LIN {X 0,Y 525.118,Z 322.281,A -85,B 0,C 180,E1 -4783.004,E2 -4783.004} C_VEL
LIN {X 0,Y 525.376,Z 308.759,A -85,B 0,C 180,E1 -4783.44,E2 -4783.44} C_VEL
LIN {X 0,Y 525.556,Z 295.266,A -85,B 0,C 180,E1 -4783.706,E2 -4783.706} C_VEL
LIN {X 0,Y 525.721,Z 203.156,A -85,B 0,C 180,E1 -4784.977,E2 -4784.977} C_VEL
LIN {X 0,Y 524.2,Z 193.139,A -85,B 0,C 180,E1 -4785.174,E2 -4785.174} C_VEL
LIN {X 0,Y 524.565,Z 174.875,A -85,B 0,C 180,E1 -4787.948,E2 -4787.948} C_VEL
LIN {X 0,Y 524.995,Z 155.161,A -85,B 0,C 180,E1 -4790.983,E2 -4790.983} C_VEL
LIN {X 0,Y 525.282,Z 140.673,A -85,B 0,C 180,E1 -4793.247,E2 -4793.247} C_VEL
LIN {X 0,Y 523.943,Z 133.222,A -85,B 0,C 180,E1 -4794.518,E2 -4794.518} C_VEL
LIN {X 0,Y 523.92,Z 133.229,A -85,B 0,C 180,E1 -4797.706,E2 -4797.706} C_VEL
LIN {X 0,Y 523.946,Z 133.218,A -85,B 0,C 180,E1 -4800.645,E2 -4800.645} C_VEL
LIN {X 0,Y 523.928,Z 133.222,A -85,B 0,C 180,E1 -4803.729,E2 -4803.729} C_VEL
LIN {X 0,Y 523.889,Z 133.223,A -85,B 0,C 180,E1 -4806.399,E2 -4806.399} C_VEL
LIN {X 0,Y 523.911,Z 133.226,A -85,B 0,C 180,E1 -4809.086,E2 -4809.086} C_VEL
LIN {X 0,Y 523.893,Z 133.223,A -85,B 0,C 180,E1 -4812.125,E2 -4812.125} C_VEL
LIN {X 0,Y 523.936,Z 133.223,A -85,B 0,C 180,E1 -4815.311,E2 -4815.311} C_VEL
LIN {X 0,Y 523.911,Z 133.225,A -85,B 0,C 180,E1 -4818.696,E2 -4818.696} C_VEL
LIN {X 0,Y 523.88,Z 133.223,A -85,B 0,C 180,E1 -4821.895,E2 -4821.895} C_VEL
LIN {X 0,Y 523.887,Z 133.228,A -85,B 0,C 180,E1 -4824.917,E2 -4824.917} C_VEL
LIN {X 0,Y 523.9,Z 133.221,A -85,B 0,C 180,E1 -4827.686,E2 -4827.686} C_VEL
LIN {X 0,Y 523.868,Z 133.227,A -85,B 0,C 180,E1 -4830.239,E2 -4830.239} C_VEL
LIN {X 0,Y 523.894,Z 133.223,A -85,B 0,C 180,E1 -4832.863,E2 -4832.863} C_VEL
LIN {X 0,Y 523.913,Z 133.221,A -85,B 0,C 180,E1 -4835.809,E2 -4835.809} C_VEL
LIN {X 0,Y 523.901,Z 133.224,A -85,B 0,C 180,E1 -4838.764,E2 -4838.764} C_VEL
LIN {X 0,Y 523.899,Z 133.22,A -85,B 0,C 180,E1 -4841.218,E2 -4841.218} C_VEL
LIN {X 0,Y 523.881,Z 133.224,A -85,B 0,C 180,E1 -4843.637,E2 -4843.637} C_VEL
LIN {X 0,Y 523.916,Z 133.226,A -85,B 0,C 180,E1 -4846.027,E2 -4846.027} C_VEL
LIN {X 0,Y 523.964,Z 133.217,A -85,B 0,C 180,E1 -4848.393,E2 -4848.393} C_VEL
LIN {X 0,Y 523.957,Z 133.216,A -85,B 0,C 180,E1 -4851.515,E2 -4851.515} C_VEL
LIN {X 0,Y 524.037,Z 133.204,A -85,B 0,C 180,E1 -4854.613,E2 -4854.613} C_VEL
LIN {X 0,Y 524.108,Z 133.2,A -85,B 0,C 180,E1 -4857.694,E2 -4857.694} C_VEL
LIN {X 0,Y 524.103,Z 133.198,A -85,B 0,C 180,E1 -4860,E2 -4860} C_VEL
LIN {X 0,Y 524.038,Z 133.205,A -85,B 0,C 180,E1 -4863.075,E2 -4863.075} C_VEL
LIN {X 0,Y 524.014,Z 133.205,A -85,B 0,C 180,E1 -4866.159,E2 -4866.159} C_VEL
LIN {X 0,Y 523.985,Z 133.218,A -85,B 0,C 180,E1 -4869.262,E2 -4869.262} C_VEL
LIN {X 0,Y 524.002,Z 133.211,A -85,B 0,C 180,E1 -4871.737,E2 -4871.737} C_VEL
LIN {X 0,Y 523.993,Z 133.214,A -85,B 0,C 180,E1 -4875.051,E2 -4875.051} C_VEL
LIN {X 0,Y 523.946,Z 133.214,A -85,B 0,C 180,E1 -4877.969,E2 -4877.969} C_VEL
LIN {X 0,Y 523.973,Z 133.214,A -85,B 0,C 180,E1 -4880.409,E2 -4880.409} C_VEL
LIN {X 0,Y 523.909,Z 133.227,A -85,B 0,C 180,E1 -4882.893,E2 -4882.893} C_VEL
LIN {X 0,Y 523.916,Z 133.221,A -85,B 0,C 180,E1 -4885.42,E2 -4885.42} C_VEL
LIN {X 0,Y 523.965,Z 133.214,A -85,B 0,C 180,E1 -4887.999,E2 -4887.999} C_VEL
LIN {X 0,Y 523.939,Z 133.223,A -85,B 0,C 180,E1 -4890.853,E2 -4890.853} C_VEL
LIN {X 0,Y 523.93,Z 133.218,A -85,B 0,C 180,E1 -4893.729,E2 -4893.729} C_VEL
LIN {X 0,Y 523.903,Z 133.23,A -85,B 0,C 180,E1 -4896.401,E2 -4896.401} C_VEL
LIN {X 0,Y 523.919,Z 133.221,A -85,B 0,C 180,E1 -4899.084,E2 -4899.084} C_VEL
LIN {X 0,Y 523.953,Z 133.222,A -85,B 0,C 180,E1 -4902.118,E2 -4902.118} C_VEL
LIN {X 0,Y 523.954,Z 133.217,A -85,B 0,C 180,E1 -4905.308,E2 -4905.308} C_VEL
LIN {X 0,Y 523.917,Z 133.222,A -85,B 0,C 180,E1 -4906.875,E2 -4906.875} C_VEL
LIN {X 0,Y 523.237,Z 133.308,A -85,B 0,C 180,E1 -4907.303,E2 -4907.303} C_VEL
LIN {X 0,Y 520.4,Z 133.666,A -85,B 0,C 180,E1 -4907.972,E2 -4907.972} C_VEL
LIN {X 0,Y 517.561,Z 134.017,A -85,B 0,C 180,E1 -4908.648,E2 -4908.648} C_VEL
LIN {X 0,Y 516.896,Z 134.098,A -85,B 0,C 180,E1 -4909.083,E2 -4909.083} C_VEL
LIN {X 0,Y 516.919,Z 134.178,A -85,B 0,C 180,E1 -4910.156,E2 -4910.156} C_VEL
LIN {X 0,Y 517.564,Z 138.657,A -85,B 0,C 180,E1 -4911.044,E2 -4911.044} C_VEL
LIN {X 0,Y 517.333,Z 154.345,A -85,B 0,C 180,E1 -4914.016,E2 -4914.016} C_VEL
LIN {X 0,Y 517.252,Z 157.921,A -85,B 0,C 180,E1 -4914.692,E2 -4914.692} C_VEL
LIN {X 0,Y 519.187,Z 168.539,A -85,B 0,C 180,E1 -4914.905,E2 -4914.905} C_VEL
LIN {X 0,Y 518.635,Z 265.409,A -85,B 0,C 180,E1 -4916.278,E2 -4916.278} C_VEL
LIN {X 0,Y 518.463,Z 278.587,A -85,B 0,C 180,E1 -4916.629,E2 -4916.629} C_VEL
LIN {X 0,Y 518.178,Z 291.605,A -85,B 0,C 180,E1 -4917.145,E2 -4917.145} C_VEL
LIN {X 0,Y 517.868,Z 303.866,A -85,B 0,C 180,E1 -4917.814,E2 -4917.814} C_VEL
LIN {X 0,Y 517.604,Z 314.805,A -85,B 0,C 180,E1 -4918.58,E2 -4918.58} C_VEL
LIN {X 0,Y 517.326,Z 325.178,A -85,B 0,C 180,E1 -4919.486,E2 -4919.486} C_VEL
LIN {X 0,Y 517.019,Z 334.784,A -85,B 0,C 180,E1 -4920.531,E2 -4920.531} C_VEL
LIN {X 0,Y 516.781,Z 343.741,A -85,B 0,C 180,E1 -4921.738,E2 -4921.738} C_VEL
LIN {X 0,Y 516.573,Z 350.564,A -85,B 0,C 180,E1 -4922.886,E2 -4922.886} C_VEL
LIN {X 0,Y 516.437,Z 356.66,A -85,B 0,C 180,E1 -4924.184,E2 -4924.184} C_VEL
LIN {X 0,Y 516.345,Z 361.243,A -85,B 0,C 180,E1 -4925.452,E2 -4925.452} C_VEL
LIN {X 0,Y 516.233,Z 364.666,A -85,B 0,C 180,E1 -4926.746,E2 -4926.746} C_VEL
LIN {X 0,Y 516.2,Z 366.557,A -85,B 0,C 180,E1 -4927.789,E2 -4927.789} C_VEL
LIN {X 0,Y 516.187,Z 368.012,A -85,B 0,C 180,E1 -4929.268,E2 -4929.268} C_VEL
LIN {X 0,Y 516.215,Z 368.215,A -85,B 0,C 180,E1 -4930.101,E2 -4930.101} C_VEL
LIN {X 0,Y 516.174,Z 367.944,A -85,B 0,C 180,E1 -4930.927,E2 -4930.927} C_VEL
LIN {X 0,Y 516.231,Z 366.456,A -85,B 0,C 180,E1 -4932.359,E2 -4932.359} C_VEL
LIN {X 0,Y 516.28,Z 363.606,A -85,B 0,C 180,E1 -4933.796,E2 -4933.796} C_VEL
LIN {X 0,Y 516.419,Z 359.814,A -85,B 0,C 180,E1 -4935.069,E2 -4935.069} C_VEL
LIN {X 0,Y 516.474,Z 355.286,A -85,B 0,C 180,E1 -4936.224,E2 -4936.224} C_VEL
LIN {X 0,Y 516.639,Z 349.277,A -85,B 0,C 180,E1 -4937.429,E2 -4937.429} C_VEL
LIN {X 0,Y 516.828,Z 341.473,A -85,B 0,C 180,E1 -4938.677,E2 -4938.677} C_VEL
LIN {X 0,Y 517.054,Z 332.52,A -85,B 0,C 180,E1 -4939.822,E2 -4939.822} C_VEL
LIN {X 0,Y 517.364,Z 322.862,A -85,B 0,C 180,E1 -4940.816,E2 -4940.816} C_VEL
LIN {X 0,Y 517.716,Z 311.758,A -85,B 0,C 180,E1 -4941.737,E2 -4941.737} C_VEL
LIN {X 0,Y 518.039,Z 300.296,A -85,B 0,C 180,E1 -4942.484,E2 -4942.484} C_VEL
LIN {X 0,Y 518.266,Z 287.201,A -85,B 0,C 180,E1 -4943.137,E2 -4943.137} C_VEL
LIN {X 0,Y 518.467,Z 274.863,A -85,B 0,C 180,E1 -4943.579,E2 -4943.579} C_VEL
LIN {X 0,Y 518.668,Z 261.95,A -85,B 0,C 180,E1 -4943.875,E2 -4943.875} C_VEL
LIN {X 0,Y 518.988,Z 167.401,A -85,B 0,C 180,E1 -4945.206,E2 -4945.206} C_VEL
LIN {X 0,Y 517.232,Z 157.733,A -85,B 0,C 180,E1 -4945.421,E2 -4945.421} C_VEL
LIN {X 0,Y 517.496,Z 141.997,A -85,B 0,C 180,E1 -4948.444,E2 -4948.444} C_VEL
LIN {X 0,Y 517.288,Z 135.99,A -85,B 0,C 180,E1 -4949.611,E2 -4949.611} C_VEL
LIN {X 0,Y 517.061,Z 134.082,A -85,B 0,C 180,E1 -4950,E2 -4950} C_VEL
LIN {X 0,Y 517.068,Z 134.08,A -85,B 0,C 180,E1 -4952.337,E2 -4952.337} C_VEL
LIN {X 0,Y 516.963,Z 134.089,A -85,B 0,C 180,E1 -4956.244,E2 -4956.244} C_VEL
LIN {X 0,Y 516.901,Z 134.095,A -85,B 0,C 180,E1 -4959.39,E2 -4959.39} C_VEL
LIN {X 0,Y 516.881,Z 134.095,A -85,B 0,C 180,E1 -4962.565,E2 -4962.565} C_VEL
LIN {X 0,Y 516.887,Z 134.096,A -85,B 0,C 180,E1 -4965.124,E2 -4965.124} C_VEL
LIN {X 0,Y 516.841,Z 134.101,A -85,B 0,C 180,E1 -4968.226,E2 -4968.226} C_VEL
LIN {X 0,Y 516.858,Z 134.098,A -85,B 0,C 180,E1 -4970.704,E2 -4970.704} C_VEL
LIN {X 0,Y 516.833,Z 134.106,A -85,B 0,C 180,E1 -4973.226,E2 -4973.226} C_VEL
LIN {X 0,Y 516.854,Z 134.099,A -85,B 0,C 180,E1 -4976.177,E2 -4976.177} C_VEL
LIN {X 0,Y 516.825,Z 134.102,A -85,B 0,C 180,E1 -4978.421,E2 -4978.421} C_VEL
LIN {X 0,Y 516.844,Z 134.106,A -85,B 0,C 180,E1 -4981.113,E2 -4981.113} C_VEL
LIN {X 0,Y 516.865,Z 134.098,A -85,B 0,C 180,E1 -4983.96,E2 -4983.96} C_VEL
LIN {X 0,Y 516.803,Z 134.108,A -85,B 0,C 180,E1 -4986.753,E2 -4986.753} C_VEL
LIN {X 0,Y 516.851,Z 134.1,A -85,B 0,C 180,E1 -4989.725,E2 -4989.725} C_VEL
LIN {X 0,Y 516.839,Z 134.107,A -85,B 0,C 180,E1 -4992.837,E2 -4992.837} C_VEL
LIN {X 0,Y 516.895,Z 134.102,A -85,B 0,C 180,E1 -4995.008,E2 -4995.008} C_VEL
LIN {X 0,Y 516.846,Z 134.102,A -85,B 0,C 180,E1 -4998.408,E2 -4998.408} C_VEL
LIN {X 0,Y 516.868,Z 134.099,A -85,B 0,C 180,E1 -5001.284,E2 -5001.284} C_VEL
LIN {X 0,Y 516.849,Z 134.108,A -85,B 0,C 180,E1 -5004.674,E2 -5004.674} C_VEL
LIN {X 0,Y 516.864,Z 134.097,A -85,B 0,C 180,E1 -5007.463,E2 -5007.463} C_VEL
LIN {X 0,Y 516.839,Z 134.108,A -85,B 0,C 180,E1 -5010.492,E2 -5010.492} C_VEL
LIN {X 0,Y 516.831,Z 134.101,A -85,B 0,C 180,E1 -5013.338,E2 -5013.338} C_VEL
LIN {X 0,Y 516.867,Z 134.099,A -85,B 0,C 180,E1 -5015.926,E2 -5015.926} C_VEL
LIN {X 0,Y 516.852,Z 134.106,A -85,B 0,C 180,E1 -5018.461,E2 -5018.461} C_VEL
LIN {X 0,Y 516.848,Z 134.1,A -85,B 0,C 180,E1 -5020.953,E2 -5020.953} C_VEL
LIN {X 0,Y 516.834,Z 134.101,A -85,B 0,C 180,E1 -5023.408,E2 -5023.408} C_VEL
LIN {X 0,Y 516.857,Z 134.102,A -85,B 0,C 180,E1 -5025.833,E2 -5025.833} C_VEL
LIN {X 0,Y 516.928,Z 134.097,A -85,B 0,C 180,E1 -5028.233,E2 -5028.233} C_VEL
LIN {X 0,Y 516.923,Z 134.091,A -85,B 0,C 180,E1 -5031.399,E2 -5031.399} C_VEL
LIN {X 0,Y 516.982,Z 134.084,A -85,B 0,C 180,E1 -5034.54,E2 -5034.54} C_VEL
LIN {X 0,Y 517.076,Z 134.076,A -85,B 0,C 180,E1 -5037.664,E2 -5037.664} C_VEL
LIN {X 0,Y 517.069,Z 134.078,A -85,B 0,C 180,E1 -5040,E2 -5040} C_VEL
LIN {X 0,Y 517.076,Z 134.073,A -85,B 0,C 180,E1 -5042.337,E2 -5042.337} C_VEL
LIN {X 0,Y 516.983,Z 134.088,A -85,B 0,C 180,E1 -5045.461,E2 -5045.461} C_VEL
LIN {X 0,Y 516.925,Z 134.09,A -85,B 0,C 180,E1 -5048.601,E2 -5048.601} C_VEL
LIN {X 0,Y 516.959,Z 134.09,A -85,B 0,C 180,E1 -5051.807,E2 -5051.807} C_VEL
LIN {X 0,Y 516.941,Z 134.092,A -85,B 0,C 180,E1 -5055.142,E2 -5055.142} C_VEL
LIN {X 0,Y 516.88,Z 134.095,A -85,B 0,C 180,E1 -5058.224,E2 -5058.224} C_VEL
LIN {X 0,Y 516.892,Z 134.095,A -85,B 0,C 180,E1 -5060.703,E2 -5060.703} C_VEL
LIN {X 0,Y 516.846,Z 134.108,A -85,B 0,C 180,E1 -5063.225,E2 -5063.225} C_VEL
LIN {X 0,Y 516.884,Z 134.095,A -85,B 0,C 180,E1 -5066.181,E2 -5066.181} C_VEL
LIN {X 0,Y 516.902,Z 134.098,A -85,B 0,C 180,E1 -5069.306,E2 -5069.306} C_VEL
LIN {X 0,Y 516.897,Z 134.096,A -85,B 0,C 180,E1 -5072.542,E2 -5072.542} C_VEL
LIN {X 0,Y 516.865,Z 134.101,A -85,B 0,C 180,E1 -5075.328,E2 -5075.328} C_VEL
LIN {X 0,Y 516.882,Z 134.095,A -85,B 0,C 180,E1 -5077.942,E2 -5077.942} C_VEL
LIN {X 0,Y 516.857,Z 134.106,A -85,B 0,C 180,E1 -5080.745,E2 -5080.745} C_VEL
LIN {X 0,Y 516.885,Z 134.095,A -85,B 0,C 180,E1 -5083.903,E2 -5083.903} C_VEL
LIN {X 0,Y 516.884,Z 134.096,A -85,B 0,C 180,E1 -5086.107,E2 -5086.107} C_VEL
LIN {X 0,Y 516.857,Z 134.099,A -85,B 0,C 180,E1 -5089.255,E2 -5089.255} C_VEL
LIN {X 0,Y 516.863,Z 134.102,A -85,B 0,C 180,E1 -5092.274,E2 -5092.274} C_VEL
LIN {X 0,Y 516.877,Z 134.096,A -85,B 0,C 180,E1 -5095.174,E2 -5095.174} C_VEL
LIN {X 0,Y 516.875,Z 134.099,A -85,B 0,C 180,E1 -5097.975,E2 -5097.975} C_VEL
LIN {X 0,Y 516.907,Z 134.097,A -85,B 0,C 180,E1 -5100.694,E2 -5100.694} C_VEL
LIN {X 0,Y 516.885,Z 134.102,A -85,B 0,C 180,E1 -5103.818,E2 -5103.818} C_VEL
LIN {X 0,Y 516.895,Z 134.142,A -85,B 0,C 180,E1 -5105.298,E2 -5105.298} C_VEL
LIN {X 0,Y 518.347,Z 142.009,A -85,B 0,C 180,E1 -5106.635,E2 -5106.635} C_VEL
LIN {X 0,Y 518.132,Z 155.153,A -85,B 0,C 180,E1 -5108.725,E2 -5108.725} C_VEL
LIN {X 0,Y 517.604,Z 176.16,A -85,B 0,C 180,E1 -5112.011,E2 -5112.011} C_VEL
LIN {X 0,Y 517.221,Z 193.048,A -85,B 0,C 180,E1 -5114.622,E2 -5114.622} C_VEL
LIN {X 0,Y 519.023,Z 205.322,A -85,B 0,C 180,E1 -5114.857,E2 -5114.857} C_VEL
LIN {X 0,Y 518.587,Z 302.204,A -85,B 0,C 180,E1 -5116.231,E2 -5116.231} C_VEL
LIN {X 0,Y 518.344,Z 315.23,A -85,B 0,C 180,E1 -5116.574,E2 -5116.574} C_VEL
LIN {X 0,Y 518.056,Z 327.837,A -85,B 0,C 180,E1 -5117.065,E2 -5117.065} C_VEL
LIN {X 0,Y 517.739,Z 340.3,A -85,B 0,C 180,E1 -5117.733,E2 -5117.733} C_VEL
LIN {X 0,Y 517.478,Z 351.993,A -85,B 0,C 180,E1 -5118.543,E2 -5118.543} C_VEL
LIN {X 0,Y 517.158,Z 362.226,A -85,B 0,C 180,E1 -5119.428,E2 -5119.428} C_VEL
LIN {X 0,Y 516.899,Z 371.429,A -85,B 0,C 180,E1 -5120.412,E2 -5120.412} C_VEL
LIN {X 0,Y 516.65,Z 380.395,A -85,B 0,C 180,E1 -5121.591,E2 -5121.591} C_VEL
LIN {X 0,Y 516.503,Z 387.613,A -85,B 0,C 180,E1 -5122.769,E2 -5122.769} C_VEL
LIN {X 0,Y 516.398,Z 394.187,A -85,B 0,C 180,E1 -5124.141,E2 -5124.141} C_VEL
LIN {X 0,Y 516.267,Z 398.532,A -85,B 0,C 180,E1 -5125.315,E2 -5125.315} C_VEL
LIN {X 0,Y 516.352,Z 400.837,A -85,B 0,C 180,E1 -5126.098,E2 -5126.098} C_VEL
LIN {X 0,Y 516.283,Z 402.7,A -85,B 0,C 180,E1 -5126.878,E2 -5126.878} C_VEL
LIN {X 0,Y 516.262,Z 404.098,A -85,B 0,C 180,E1 -5127.659,E2 -5127.659} C_VEL
LIN {X 0,Y 516.166,Z 405.7,A -85,B 0,C 180,E1 -5129.22,E2 -5129.22} C_VEL
LIN {X 0,Y 516.164,Z 405.915,A -85,B 0,C 180,E1 -5130,E2 -5130} C_VEL
LIN {X 0,Y 516.192,Z 405.088,A -85,B 0,C 180,E1 -5131.56,E2 -5131.56} C_VEL
LIN {X 0,Y 516.262,Z 404.09,A -85,B 0,C 180,E1 -5132.34,E2 -5132.34} C_VEL
LIN {X 0,Y 516.283,Z 402.689,A -85,B 0,C 180,E1 -5133.121,E2 -5133.121} C_VEL
LIN {X 0,Y 516.31,Z 399.743,A -85,B 0,C 180,E1 -5134.293,E2 -5134.293} C_VEL
LIN {X 0,Y 516.367,Z 395.755,A -85,B 0,C 180,E1 -5135.467,E2 -5135.467} C_VEL
LIN {X 0,Y 516.405,Z 390.603,A -85,B 0,C 180,E1 -5136.647,E2 -5136.647} C_VEL
LIN {X 0,Y 516.535,Z 384.161,A -85,B 0,C 180,E1 -5137.82,E2 -5137.82} C_VEL
LIN {X 0,Y 516.748,Z 376.105,A -85,B 0,C 180,E1 -5138.998,E2 -5138.998} C_VEL
LIN {X 0,Y 516.942,Z 367.894,A -85,B 0,C 180,E1 -5139.982,E2 -5139.982} C_VEL
LIN {X 0,Y 517.274,Z 357.886,A -85,B 0,C 180,E1 -5140.965,E2 -5140.965} C_VEL
LIN {X 0,Y 517.569,Z 348.006,A -85,B 0,C 180,E1 -5141.752,E2 -5141.752} C_VEL
LIN {X 0,Y 517.842,Z 336.853,A -85,B 0,C 180,E1 -5142.465,E2 -5142.465} C_VEL
LIN {X 0,Y 518.125,Z 324.348,A -85,B 0,C 180,E1 -5143.082,E2 -5143.082} C_VEL
LIN {X 0,Y 518.413,Z 311.185,A -85,B 0,C 180,E1 -5143.549,E2 -5143.549} C_VEL
LIN {X 0,Y 518.658,Z 297.998,A -85,B 0,C 180,E1 -5143.842,E2 -5143.842} C_VEL
LIN {X 0,Y 518.972,Z 204.59,A -85,B 0,C 180,E1 -5145.153,E2 -5145.153} C_VEL
LIN {X 0,Y 517.217,Z 192.867,A -85,B 0,C 180,E1 -5145.383,E2 -5145.383} C_VEL
LIN {X 0,Y 517.669,Z 173.316,A -85,B 0,C 180,E1 -5148.4,E2 -5148.4} C_VEL
LIN {X 0,Y 518.065,Z 154.915,A -85,B 0,C 180,E1 -5151.278,E2 -5151.278} C_VEL
LIN {X 0,Y 518.322,Z 141.743,A -85,B 0,C 180,E1 -5153.366,E2 -5153.366} C_VEL
LIN {X 0,Y 516.882,Z 134.101,A -85,B 0,C 180,E1 -5154.697,E2 -5154.697} C_VEL
LIN {X 0,Y 516.877,Z 134.105,A -85,B 0,C 180,E1 -5157.536,E2 -5157.536} C_VEL
LIN {X 0,Y 516.869,Z 134.102,A -85,B 0,C 180,E1 -5160.205,E2 -5160.205} C_VEL
LIN {X 0,Y 516.883,Z 134.098,A -85,B 0,C 180,E1 -5162.948,E2 -5162.948} C_VEL
LIN {X 0,Y 516.858,Z 134.103,A -85,B 0,C 180,E1 -5165.782,E2 -5165.782} C_VEL
LIN {X 0,Y 516.876,Z 134.099,A -85,B 0,C 180,E1 -5168.716,E2 -5168.716} C_VEL
LIN {X 0,Y 516.845,Z 134.102,A -85,B 0,C 180,E1 -5171.782,E2 -5171.782} C_VEL
LIN {X 0,Y 516.898,Z 134.1,A -85,B 0,C 180,E1 -5175.007,E2 -5175.007} C_VEL
LIN {X 0,Y 516.849,Z 134.102,A -85,B 0,C 180,E1 -5178.407,E2 -5178.407} C_VEL
LIN {X 0,Y 516.857,Z 134.101,A -85,B 0,C 180,E1 -5181.282,E2 -5181.282} C_VEL
LIN {X 0,Y 516.827,Z 134.11,A -85,B 0,C 180,E1 -5184.677,E2 -5184.677} C_VEL
LIN {X 0,Y 516.865,Z 134.098,A -85,B 0,C 180,E1 -5187.463,E2 -5187.463} C_VEL
LIN {X 0,Y 516.84,Z 134.106,A -85,B 0,C 180,E1 -5190.491,E2 -5190.491} C_VEL
LIN {X 0,Y 516.831,Z 134.099,A -85,B 0,C 180,E1 -5193.337,E2 -5193.337} C_VEL
LIN {X 0,Y 516.868,Z 134.099,A -85,B 0,C 180,E1 -5195.925,E2 -5195.925} C_VEL
LIN {X 0,Y 516.852,Z 134.106,A -85,B 0,C 180,E1 -5198.46,E2 -5198.46} C_VEL
LIN {X 0,Y 516.848,Z 134.099,A -85,B 0,C 180,E1 -5200.952,E2 -5200.952} C_VEL
LIN {X 0,Y 516.837,Z 134.1,A -85,B 0,C 180,E1 -5203.407,E2 -5203.407} C_VEL
LIN {X 0,Y 516.874,Z 134.101,A -85,B 0,C 180,E1 -5205.833,E2 -5205.833} C_VEL
LIN {X 0,Y 516.929,Z 134.095,A -85,B 0,C 180,E1 -5208.232,E2 -5208.232} C_VEL
LIN {X 0,Y 516.933,Z 134.089,A -85,B 0,C 180,E1 -5211.399,E2 -5211.399} C_VEL
LIN {X 0,Y 516.988,Z 134.082,A -85,B 0,C 180,E1 -5214.539,E2 -5214.539} C_VEL
LIN {X 0,Y 517.077,Z 134.075,A -85,B 0,C 180,E1 -5217.663,E2 -5217.663} C_VEL
LIN {X 0,Y 517.072,Z 134.073,A -85,B 0,C 180,E1 -5220,E2 -5220} C_VEL
LIN {X 0,Y 517.082,Z 134.07,A -85,B 0,C 180,E1 -5222.336,E2 -5222.336} C_VEL
LIN {X 0,Y 517.015,Z 134.084,A -85,B 0,C 180,E1 -5225.46,E2 -5225.46} C_VEL
LIN {X 0,Y 516.956,Z 134.087,A -85,B 0,C 180,E1 -5228.6,E2 -5228.6} C_VEL
LIN {X 0,Y 516.955,Z 134.089,A -85,B 0,C 180,E1 -5231.806,E2 -5231.806} C_VEL
LIN {X 0,Y 516.945,Z 134.093,A -85,B 0,C 180,E1 -5235.145,E2 -5235.145} C_VEL
LIN {X 0,Y 516.914,Z 134.09,A -85,B 0,C 180,E1 -5238.222,E2 -5238.222} C_VEL
LIN {X 0,Y 516.914,Z 134.097,A -85,B 0,C 180,E1 -5240.701,E2 -5240.701} C_VEL
LIN {X 0,Y 516.887,Z 134.096,A -85,B 0,C 180,E1 -5244.073,E2 -5244.073} C_VEL
LIN {X 0,Y 516.909,Z 134.1,A -85,B 0,C 180,E1 -5246.658,E2 -5246.658} C_VEL
LIN {X 0,Y 516.91,Z 134.093,A -85,B 0,C 180,E1 -5249.523,E2 -5249.523} C_VEL
LIN {X 0,Y 516.894,Z 134.102,A -85,B 0,C 180,E1 -5252.542,E2 -5252.542} C_VEL
LIN {X 0,Y 516.865,Z 134.099,A -85,B 0,C 180,E1 -5255.329,E2 -5255.329} C_VEL
LIN {X 0,Y 516.88,Z 134.101,A -85,B 0,C 180,E1 -5257.943,E2 -5257.943} C_VEL
LIN {X 0,Y 516.883,Z 134.102,A -85,B 0,C 180,E1 -5260.741,E2 -5260.741} C_VEL
LIN {X 0,Y 516.883,Z 134.101,A -85,B 0,C 180,E1 -5262.831,E2 -5262.831} C_VEL
LIN {X 0,Y 516.921,Z 134.093,A -85,B 0,C 180,E1 -5265.01,E2 -5265.01} C_VEL
LIN {X 0,Y 516.92,Z 134.099,A -85,B 0,C 180,E1 -5268.397,E2 -5268.397} C_VEL
LIN {X 0,Y 516.896,Z 134.098,A -85,B 0,C 180,E1 -5269.083,E2 -5269.083} C_VEL
LIN {X 0,Y 516.614,Z 134.436,A -85,B 0,C 180,E1 -5269.514,E2 -5269.514} C_VEL
LIN {X 0,Y 515.402,Z 135.953,A -85,B 0,C 180,E1 -5270.133,E2 -5270.133} C_VEL
LIN {X 0,Y 513.73,Z 138.303,A -85,B 0,C 180,E1 -5270.715,E2 -5270.715} C_VEL
LIN {X 0,Y 511.118,Z 143.341,A -85,B 0,C 180,E1 -5271.664,E2 -5271.664} C_VEL
LIN {X 0,Y 510.504,Z 146.494,A -85,B 0,C 180,E1 -5272.245,E2 -5272.245} C_VEL
LIN {X 0,Y 510.306,Z 158.072,A -85,B 0,C 180,E1 -5274.459,E2 -5274.459} C_VEL
LIN {X 0,Y 512.366,Z 169.773,A -85,B 0,C 180,E1 -5274.707,E2 -5274.707} C_VEL
LIN {X 0,Y 511.749,Z 265.725,A -85,B 0,C 180,E1 -5276.088,E2 -5276.088} C_VEL
LIN {X 0,Y 511.592,Z 278.907,A -85,B 0,C 180,E1 -5276.446,E2 -5276.446} C_VEL
LIN {X 0,Y 511.325,Z 290.944,A -85,B 0,C 180,E1 -5276.925,E2 -5276.925} C_VEL
LIN {X 0,Y 510.997,Z 302.796,A -85,B 0,C 180,E1 -5277.562,E2 -5277.562} C_VEL
LIN {X 0,Y 510.693,Z 314.179,A -85,B 0,C 180,E1 -5278.354,E2 -5278.354} C_VEL
LIN {X 0,Y 510.341,Z 324.531,A -85,B 0,C 180,E1 -5279.252,E2 -5279.252} C_VEL
LIN {X 0,Y 510.044,Z 333.919,A -85,B 0,C 180,E1 -5280.261,E2 -5280.261} C_VEL
LIN {X 0,Y 509.807,Z 342.295,A -85,B 0,C 180,E1 -5281.371,E2 -5281.371} C_VEL
LIN {X 0,Y 509.539,Z 350.381,A -85,B 0,C 180,E1 -5282.702,E2 -5282.702} C_VEL
LIN {X 0,Y 509.409,Z 355.672,A -85,B 0,C 180,E1 -5283.801,E2 -5283.801} C_VEL
LIN {X 0,Y 509.284,Z 360.635,A -85,B 0,C 180,E1 -5285.109,E2 -5285.109} C_VEL
LIN {X 0,Y 509.165,Z 364.264,A -85,B 0,C 180,E1 -5286.404,E2 -5286.404} C_VEL
LIN {X 0,Y 509.126,Z 366.661,A -85,B 0,C 180,E1 -5287.647,E2 -5287.647} C_VEL
LIN {X 0,Y 509.084,Z 368.098,A -85,B 0,C 180,E1 -5288.965,E2 -5288.965} C_VEL
LIN {X 0,Y 509.142,Z 368.441,A -85,B 0,C 180,E1 -5289.824,E2 -5289.824} C_VEL
LIN {X 0,Y 509.107,Z 368.36,A -85,B 0,C 180,E1 -5290.652,E2 -5290.652} C_VEL
LIN {X 0,Y 509.09,Z 367.803,A -85,B 0,C 180,E1 -5291.487,E2 -5291.487} C_VEL
LIN {X 0,Y 509.149,Z 366.812,A -85,B 0,C 180,E1 -5292.322,E2 -5292.322} C_VEL
LIN {X 0,Y 509.17,Z 365.409,A -85,B 0,C 180,E1 -5293.15,E2 -5293.15} C_VEL
LIN {X 0,Y 509.272,Z 362.418,A -85,B 0,C 180,E1 -5294.389,E2 -5294.389} C_VEL
LIN {X 0,Y 509.364,Z 358.35,A -85,B 0,C 180,E1 -5295.62,E2 -5295.62} C_VEL
LIN {X 0,Y 509.491,Z 352.07,A -85,B 0,C 180,E1 -5297.047,E2 -5297.047} C_VEL
LIN {X 0,Y 509.728,Z 344.555,A -85,B 0,C 180,E1 -5298.373,E2 -5298.373} C_VEL
LIN {X 0,Y 509.954,Z 336.705,A -85,B 0,C 180,E1 -5299.478,E2 -5299.478} C_VEL
LIN {X 0,Y 510.244,Z 327.934,A -85,B 0,C 180,E1 -5300.486,E2 -5300.486} C_VEL
LIN {X 0,Y 510.609,Z 317.147,A -85,B 0,C 180,E1 -5301.491,E2 -5301.491} C_VEL
LIN {X 0,Y 510.951,Z 306.184,A -85,B 0,C 180,E1 -5302.305,E2 -5302.305} C_VEL
LIN {X 0,Y 511.239,Z 294.331,A -85,B 0,C 180,E1 -5302.992,E2 -5302.992} C_VEL
LIN {X 0,Y 511.488,Z 281.76,A -85,B 0,C 180,E1 -5303.541,E2 -5303.541} C_VEL
LIN {X 0,Y 511.677,Z 269.483,A -85,B 0,C 180,E1 -5303.914,E2 -5303.914} C_VEL
LIN {X 0,Y 511.808,Z 253.936,A -85,B 0,C 180,E1 -5304.188,E2 -5304.188} C_VEL
LIN {X 0,Y 512.187,Z 168.281,A -85,B 0,C 180,E1 -5305.401,E2 -5305.401} C_VEL
LIN {X 0,Y 510.226,Z 157.991,A -85,B 0,C 180,E1 -5305.631,E2 -5305.631} C_VEL
LIN {X 0,Y 510.53,Z 142.538,A -85,B 0,C 180,E1 -5308.62,E2 -5308.62} C_VEL
LIN {X 0,Y 510.122,Z 135.549,A -85,B 0,C 180,E1 -5310,E2 -5310} C_VEL
LIN {X 0,Y 509.989,Z 134.963,A -85,B 0,C 180,E1 -5310.148,E2 -5310.148} C_VEL
LIN {X 0,Y 510.036,Z 134.955,A -85,B 0,C 180,E1 -5312.369,E2 -5312.369} C_VEL
LIN {X 0,Y 509.93,Z 134.964,A -85,B 0,C 180,E1 -5315.536,E2 -5315.536} C_VEL
LIN {X 0,Y 509.869,Z 134.977,A -85,B 0,C 180,E1 -5317.923,E2 -5317.923} C_VEL
LIN {X 0,Y 509.857,Z 134.971,A -85,B 0,C 180,E1 -5321.127,E2 -5321.127} C_VEL
LIN {X 0,Y 509.814,Z 134.981,A -85,B 0,C 180,E1 -5323.554,E2 -5323.554} C_VEL
LIN {X 0,Y 509.787,Z 134.983,A -85,B 0,C 180,E1 -5326.005,E2 -5326.005} C_VEL
LIN {X 0,Y 509.803,Z 134.977,A -85,B 0,C 180,E1 -5328.486,E2 -5328.486} C_VEL
LIN {X 0,Y 509.808,Z 134.978,A -85,B 0,C 180,E1 -5331.004,E2 -5331.004} C_VEL
LIN {X 0,Y 509.793,Z 134.986,A -85,B 0,C 180,E1 -5333.566,E2 -5333.566} C_VEL
LIN {X 0,Y 509.795,Z 134.978,A -85,B 0,C 180,E1 -5336.353,E2 -5336.353} C_VEL
LIN {X 0,Y 509.789,Z 134.981,A -85,B 0,C 180,E1 -5338.85,E2 -5338.85} C_VEL
LIN {X 0,Y 509.784,Z 134.984,A -85,B 0,C 180,E1 -5341.593,E2 -5341.593} C_VEL
LIN {X 0,Y 509.818,Z 134.975,A -85,B 0,C 180,E1 -5344.417,E2 -5344.417} C_VEL
LIN {X 0,Y 509.771,Z 134.987,A -85,B 0,C 180,E1 -5347.345,E2 -5347.345} C_VEL
LIN {X 0,Y 509.792,Z 134.979,A -85,B 0,C 180,E1 -5350.387,E2 -5350.387} C_VEL
LIN {X 0,Y 509.79,Z 134.98,A -85,B 0,C 180,E1 -5353.576,E2 -5353.576} C_VEL
LIN {X 0,Y 509.791,Z 134.981,A -85,B 0,C 180,E1 -5356.426,E2 -5356.426} C_VEL
LIN {X 0,Y 509.811,Z 134.976,A -85,B 0,C 180,E1 -5359.616,E2 -5359.616} C_VEL
LIN {X 0,Y 509.782,Z 134.987,A -85,B 0,C 180,E1 -5362.657,E2 -5362.657} C_VEL
LIN {X 0,Y 509.831,Z 134.973,A -85,B 0,C 180,E1 -5365.803,E2 -5365.803} C_VEL
LIN {X 0,Y 509.815,Z 134.982,A -85,B 0,C 180,E1 -5368.727,E2 -5368.727} C_VEL
LIN {X 0,Y 509.823,Z 134.977,A -85,B 0,C 180,E1 -5372.051,E2 -5372.051} C_VEL
LIN {X 0,Y 509.788,Z 134.984,A -85,B 0,C 180,E1 -5374.7,E2 -5374.7} C_VEL
LIN {X 0,Y 509.826,Z 134.974,A -85,B 0,C 180,E1 -5377.46,E2 -5377.46} C_VEL
LIN {X 0,Y 509.809,Z 134.98,A -85,B 0,C 180,E1 -5380.68,E2 -5380.68} C_VEL
LIN {X 0,Y 509.79,Z 134.978,A -85,B 0,C 180,E1 -5383.172,E2 -5383.172} C_VEL
LIN {X 0,Y 509.822,Z 134.976,A -85,B 0,C 180,E1 -5385.633,E2 -5385.633} C_VEL
LIN {X 0,Y 509.893,Z 134.975,A -85,B 0,C 180,E1 -5388.132,E2 -5388.132} C_VEL
LIN {X 0,Y 509.876,Z 134.968,A -85,B 0,C 180,E1 -5391.28,E2 -5391.28} C_VEL
LIN {X 0,Y 509.919,Z 134.966,A -85,B 0,C 180,E1 -5393.67,E2 -5393.67} C_VEL
LIN {X 0,Y 509.886,Z 134.966,A -85,B 0,C 180,E1 -5396.84,E2 -5396.84} C_VEL
LIN {X 0,Y 509.925,Z 134.963,A -85,B 0,C 180,E1 -5398.421,E2 -5398.421} C_VEL
LIN {X 0,Y 510.038,Z 134.954,A -85,B 0,C 180,E1 -5400,E2 -5400} C_VEL
LIN {X 0,Y 510.044,Z 134.948,A -85,B 0,C 180,E1 -5402.37,E2 -5402.37} C_VEL
LIN {X 0,Y 509.936,Z 134.967,A -85,B 0,C 180,E1 -5405.537,E2 -5405.537} C_VEL
LIN {X 0,Y 509.88,Z 134.972,A -85,B 0,C 180,E1 -5407.923,E2 -5407.923} C_VEL
LIN {X 0,Y 509.916,Z 134.966,A -85,B 0,C 180,E1 -5411.126,E2 -5411.126} C_VEL
LIN {X 0,Y 509.845,Z 134.972,A -85,B 0,C 180,E1 -5414.367,E2 -5414.367} C_VEL
LIN {X 0,Y 509.801,Z 134.979,A -85,B 0,C 180,E1 -5416.828,E2 -5416.828} C_VEL
LIN {X 0,Y 509.849,Z 134.98,A -85,B 0,C 180,E1 -5419.319,E2 -5419.319} C_VEL
LIN {X 0,Y 509.812,Z 134.977,A -85,B 0,C 180,E1 -5421.852,E2 -5421.852} C_VEL
LIN {X 0,Y 509.831,Z 134.974,A -85,B 0,C 180,E1 -5424.52,E2 -5424.52} C_VEL
LIN {X 0,Y 509.823,Z 134.982,A -85,B 0,C 180,E1 -5427.06,E2 -5427.06} C_VEL
LIN {X 0,Y 509.83,Z 134.974,A -85,B 0,C 180,E1 -5429.753,E2 -5429.753} C_VEL
LIN {X 0,Y 509.849,Z 134.976,A -85,B 0,C 180,E1 -5432.769,E2 -5432.769} C_VEL
LIN {X 0,Y 509.825,Z 134.975,A -85,B 0,C 180,E1 -5435.577,E2 -5435.577} C_VEL
LIN {X 0,Y 509.852,Z 134.973,A -85,B 0,C 180,E1 -5438.338,E2 -5438.338} C_VEL
LIN {X 0,Y 509.812,Z 134.977,A -85,B 0,C 180,E1 -5441.43,E2 -5441.43} C_VEL
LIN {X 0,Y 509.844,Z 134.98,A -85,B 0,C 180,E1 -5444.67,E2 -5444.67} C_VEL
LIN {X 0,Y 509.795,Z 134.978,A -85,B 0,C 180,E1 -5447.506,E2 -5447.506} C_VEL
LIN {X 0,Y 509.836,Z 134.981,A -85,B 0,C 180,E1 -5450.646,E2 -5450.646} C_VEL
LIN {X 0,Y 509.812,Z 134.976,A -85,B 0,C 180,E1 -5453.645,E2 -5453.645} C_VEL
LIN {X 0,Y 509.843,Z 134.979,A -85,B 0,C 180,E1 -5456.537,E2 -5456.537} C_VEL
LIN {X 0,Y 509.838,Z 134.974,A -85,B 0,C 180,E1 -5459.333,E2 -5459.333} C_VEL
LIN {X 0,Y 509.836,Z 134.98,A -85,B 0,C 180,E1 -5462.051,E2 -5462.051} C_VEL
LIN {X 0,Y 509.858,Z 135.038,A -85,B 0,C 180,E1 -5465.132,E2 -5465.132} C_VEL
LIN {X 0,Y 511.355,Z 143.055,A -85,B 0,C 180,E1 -5466.511,E2 -5466.511} C_VEL
LIN {X 0,Y 511.28,Z 152.255,A -85,B 0,C 180,E1 -5468.002,E2 -5468.002} C_VEL
LIN {X 0,Y 510.799,Z 167.995,A -85,B 0,C 180,E1 -5470.509,E2 -5470.509} C_VEL
LIN {X 0,Y 510.398,Z 186.329,A -85,B 0,C 180,E1 -5473.398,E2 -5473.398} C_VEL
LIN {X 0,Y 510.232,Z 192.786,A -85,B 0,C 180,E1 -5474.406,E2 -5474.406} C_VEL
LIN {X 0,Y 512.167,Z 207.134,A -85,B 0,C 180,E1 -5474.679,E2 -5474.679} C_VEL
LIN {X 0,Y 511.694,Z 301.891,A -85,B 0,C 180,E1 -5476.041,E2 -5476.041} C_VEL
LIN {X 0,Y 511.448,Z 314.935,A -85,B 0,C 180,E1 -5476.389,E2 -5476.389} C_VEL
LIN {X 0,Y 511.123,Z 327.553,A -85,B 0,C 180,E1 -5476.887,E2 -5476.887} C_VEL
LIN {X 0,Y 510.815,Z 339.325,A -85,B 0,C 180,E1 -5477.52,E2 -5477.52} C_VEL
LIN {X 0,Y 510.505,Z 350.423,A -85,B 0,C 180,E1 -5478.284,E2 -5478.284} C_VEL
LIN {X 0,Y 510.203,Z 360.905,A -85,B 0,C 180,E1 -5479.182,E2 -5479.182} C_VEL
LIN {X 0,Y 509.88,Z 369.473,A -85,B 0,C 180,E1 -5480.078,E2 -5480.078} C_VEL
LIN {X 0,Y 509.649,Z 377.381,A -85,B 0,C 180,E1 -5481.075,E2 -5481.075} C_VEL
LIN {X 0,Y 509.46,Z 385.106,A -85,B 0,C 180,E1 -5482.27,E2 -5482.27} C_VEL
LIN {X 0,Y 509.289,Z 392.221,A -85,B 0,C 180,E1 -5483.662,E2 -5483.662} C_VEL
LIN {X 0,Y 509.241,Z 396.958,A -85,B 0,C 180,E1 -5484.853,E2 -5484.853} C_VEL
LIN {X 0,Y 509.245,Z 400.577,A -85,B 0,C 180,E1 -5486.043,E2 -5486.043} C_VEL
LIN {X 0,Y 509.201,Z 402.442,A -85,B 0,C 180,E1 -5486.835,E2 -5486.835} C_VEL
LIN {X 0,Y 509.19,Z 403.841,A -85,B 0,C 180,E1 -5487.627,E2 -5487.627} C_VEL
LIN {X 0,Y 509.079,Z 405.442,A -85,B 0,C 180,E1 -5489.209,E2 -5489.209} C_VEL
LIN {X 0,Y 509.075,Z 405.656,A -85,B 0,C 180,E1 -5490,E2 -5490} C_VEL
LIN {X 0,Y 509.113,Z 404.828,A -85,B 0,C 180,E1 -5491.582,E2 -5491.582} C_VEL
LIN {X 0,Y 509.19,Z 403.83,A -85,B 0,C 180,E1 -5492.373,E2 -5492.373} C_VEL
LIN {X 0,Y 509.201,Z 402.427,A -85,B 0,C 180,E1 -5493.165,E2 -5493.165} C_VEL
LIN {X 0,Y 509.202,Z 399.478,A -85,B 0,C 180,E1 -5494.353,E2 -5494.353} C_VEL
LIN {X 0,Y 509.282,Z 395.489,A -85,B 0,C 180,E1 -5495.543,E2 -5495.543} C_VEL
LIN {X 0,Y 509.365,Z 389.455,A -85,B 0,C 180,E1 -5496.914,E2 -5496.914} C_VEL
LIN {X 0,Y 509.494,Z 382.648,A -85,B 0,C 180,E1 -5498.128,E2 -5498.128} C_VEL
LIN {X 0,Y 509.729,Z 374.333,A -85,B 0,C 180,E1 -5499.323,E2 -5499.323} C_VEL
LIN {X 0,Y 509.967,Z 365.806,A -85,B 0,C 180,E1 -5500.321,E2 -5500.321} C_VEL
LIN {X 0,Y 510.334,Z 355.275,A -85,B 0,C 180,E1 -5501.317,E2 -5501.317} C_VEL
LIN {X 0,Y 510.645,Z 344.22,A -85,B 0,C 180,E1 -5502.16,E2 -5502.16} C_VEL
LIN {X 0,Y 510.984,Z 333.43,A -85,B 0,C 180,E1 -5502.814,E2 -5502.814} C_VEL
LIN {X 0,Y 511.254,Z 321.67,A -85,B 0,C 180,E1 -5503.363,E2 -5503.363} C_VEL
LIN {X 0,Y 511.572,Z 308.143,A -85,B 0,C 180,E1 -5503.81,E2 -5503.81} C_VEL
LIN {X 0,Y 511.801,Z 294.61,A -85,B 0,C 180,E1 -5504.082,E2 -5504.082} C_VEL
LIN {X 0,Y 512.011,Z 204.725,A -85,B 0,C 180,E1 -5505.361,E2 -5505.361} C_VEL
LIN {X 0,Y 510.208,Z 192.569,A -85,B 0,C 180,E1 -5505.608,E2 -5505.608} C_VEL
LIN {X 0,Y 510.704,Z 173.073,A -85,B 0,C 180,E1 -5508.66,E2 -5508.66} C_VEL
LIN {X 0,Y 511.114,Z 155.986,A -85,B 0,C 180,E1 -5511.37,E2 -5511.37} C_VEL
LIN {X 0,Y 511.469,Z 144.772,A -85,B 0,C 180,E1 -5513.167,E2 -5513.167} C_VEL
LIN {X 0,Y 510.355,Z 137.556,A -85,B 0,C 180,E1 -5514.401,E2 -5514.401} C_VEL
LIN {X 0,Y 509.823,Z 134.981,A -85,B 0,C 180,E1 -5514.888,E2 -5514.888} C_VEL
LIN {X 0,Y 509.826,Z 134.979,A -85,B 0,C 180,E1 -5517.059,E2 -5517.059} C_VEL
LIN {X 0,Y 509.854,Z 134.979,A -85,B 0,C 180,E1 -5519.751,E2 -5519.751} C_VEL
LIN {X 0,Y 509.847,Z 134.974,A -85,B 0,C 180,E1 -5522.769,E2 -5522.769} C_VEL
LIN {X 0,Y 509.816,Z 134.983,A -85,B 0,C 180,E1 -5525.576,E2 -5525.576} C_VEL
LIN {X 0,Y 509.822,Z 134.976,A -85,B 0,C 180,E1 -5528.341,E2 -5528.341} C_VEL
LIN {X 0,Y 509.804,Z 134.983,A -85,B 0,C 180,E1 -5531.431,E2 -5531.431} C_VEL
LIN {X 0,Y 509.842,Z 134.975,A -85,B 0,C 180,E1 -5534.67,E2 -5534.67} C_VEL
LIN {X 0,Y 509.79,Z 134.982,A -85,B 0,C 180,E1 -5537.505,E2 -5537.505} C_VEL
LIN {X 0,Y 509.818,Z 134.98,A -85,B 0,C 180,E1 -5540.645,E2 -5540.645} C_VEL
LIN {X 0,Y 509.76,Z 134.983,A -85,B 0,C 180,E1 -5543.641,E2 -5543.641} C_VEL
LIN {X 0,Y 509.824,Z 134.978,A -85,B 0,C 180,E1 -5546.536,E2 -5546.536} C_VEL
LIN {X 0,Y 509.803,Z 134.976,A -85,B 0,C 180,E1 -5549.331,E2 -5549.331} C_VEL
LIN {X 0,Y 509.824,Z 134.976,A -85,B 0,C 180,E1 -5552.05,E2 -5552.05} C_VEL
LIN {X 0,Y 509.788,Z 134.984,A -85,B 0,C 180,E1 -5554.699,E2 -5554.699} C_VEL
LIN {X 0,Y 509.827,Z 134.97,A -85,B 0,C 180,E1 -5557.459,E2 -5557.459} C_VEL
LIN {X 0,Y 509.81,Z 134.978,A -85,B 0,C 180,E1 -5560.679,E2 -5560.679} C_VEL
LIN {X 0,Y 509.792,Z 134.978,A -85,B 0,C 180,E1 -5563.171,E2 -5563.171} C_VEL
LIN {X 0,Y 509.848,Z 134.974,A -85,B 0,C 180,E1 -5565.633,E2 -5565.633} C_VEL
LIN {X 0,Y 509.893,Z 134.973,A -85,B 0,C 180,E1 -5568.13,E2 -5568.13} C_VEL
LIN {X 0,Y 509.887,Z 134.966,A -85,B 0,C 180,E1 -5571.279,E2 -5571.279} C_VEL
LIN {X 0,Y 509.943,Z 134.96,A -85,B 0,C 180,E1 -5574.463,E2 -5574.463} C_VEL
LIN {X 0,Y 510.046,Z 134.95,A -85,B 0,C 180,E1 -5577.63,E2 -5577.63} C_VEL
LIN {X 0,Y 510.041,Z 134.949,A -85,B 0,C 180,E1 -5580,E2 -5580} C_VEL
LIN {X 0,Y 510.052,Z 134.945,A -85,B 0,C 180,E1 -5582.369,E2 -5582.369} C_VEL
LIN {X 0,Y 509.966,Z 134.961,A -85,B 0,C 180,E1 -5585.535,E2 -5585.535} C_VEL
LIN {X 0,Y 509.905,Z 134.966,A -85,B 0,C 180,E1 -5588.72,E2 -5588.72} C_VEL
LIN {X 0,Y 509.907,Z 134.966,A -85,B 0,C 180,E1 -5591.931,E2 -5591.931} C_VEL
LIN {X 0,Y 509.897,Z 134.972,A -85,B 0,C 180,E1 -5595.241,E2 -5595.241} C_VEL
LIN {X 0,Y 509.859,Z 134.971,A -85,B 0,C 180,E1 -5598.483,E2 -5598.483} C_VEL
LIN {X 0,Y 509.851,Z 134.978,A -85,B 0,C 180,E1 -5601.001,E2 -5601.001} C_VEL
LIN {X 0,Y 509.82,Z 134.977,A -85,B 0,C 180,E1 -5603.563,E2 -5603.563} C_VEL
LIN {X 0,Y 509.887,Z 134.97,A -85,B 0,C 180,E1 -5606.372,E2 -5606.372} C_VEL
LIN {X 0,Y 509.875,Z 134.976,A -85,B 0,C 180,E1 -5608.844,E2 -5608.844} C_VEL
LIN {X 0,Y 509.819,Z 134.976,A -85,B 0,C 180,E1 -5611.59,E2 -5611.59} C_VEL
LIN {X 0,Y 509.838,Z 134.981,A -85,B 0,C 180,E1 -5614.414,E2 -5614.414} C_VEL
LIN {X 0,Y 509.816,Z 134.978,A -85,B 0,C 180,E1 -5617.34,E2 -5617.34} C_VEL
LIN {X 0,Y 509.837,Z 134.984,A -85,B 0,C 180,E1 -5620.382,E2 -5620.382} C_VEL
LIN {X 0,Y 509.823,Z 134.979,A -85,B 0,C 180,E1 -5623.062,E2 -5623.062} C_VEL
LIN {X 0,Y 509.829,Z 134.98,A -85,B 0,C 180,E1 -5625.792,E2 -5625.792} C_VEL
LIN {X 0,Y 509.864,Z 134.977,A -85,B 0,C 180,E1 -5628.575,E2 -5628.575} C_VEL
LIN {X 0,Y 509.909,Z 135.045,A -85,B 0,C 180,E1 -5630.017,E2 -5630.017} C_VEL
LIN {X 0,Y 510.619,Z 139.876,A -85,B 0,C 180,E1 -5630.973,E2 -5630.973} C_VEL
LIN {X 0,Y 510.504,Z 146.494,A -85,B 0,C 180,E1 -5632.245,E2 -5632.245} C_VEL
LIN {X 0,Y 509.813,Z 148.581,A -85,B 0,C 180,E1 -5632.617,E2 -5632.617} C_VEL
LIN {X 0,Y 506.931,Z 152.106,A -85,B 0,C 180,E1 -5633.178,E2 -5633.178} C_VEL
LIN {X 0,Y 504.031,Z 155.644,A -85,B 0,C 180,E1 -5633.744,E2 -5633.744} C_VEL
LIN {X 0,Y 503.328,Z 157.735,A -85,B 0,C 180,E1 -5634.122,E2 -5634.122} C_VEL
LIN {X 0,Y 503.321,Z 158.37,A -85,B 0,C 180,E1 -5634.244,E2 -5634.244} C_VEL
LIN {X 0,Y 505.529,Z 170.107,A -85,B 0,C 180,E1 -5634.49,E2 -5634.49} C_VEL
LIN {X 0,Y 504.925,Z 264.912,A -85,B 0,C 180,E1 -5635.868,E2 -5635.868} C_VEL
LIN {X 0,Y 504.717,Z 278.066,A -85,B 0,C 180,E1 -5636.216,E2 -5636.216} C_VEL
LIN {X 0,Y 504.469,Z 290.508,A -85,B 0,C 180,E1 -5636.707,E2 -5636.707} C_VEL
LIN {X 0,Y 504.157,Z 301.763,A -85,B 0,C 180,E1 -5637.304,E2 -5637.304} C_VEL
LIN {X 0,Y 503.772,Z 313.317,A -85,B 0,C 180,E1 -5638.098,E2 -5638.098} C_VEL
LIN {X 0,Y 503.4,Z 323.926,A -85,B 0,C 180,E1 -5639.015,E2 -5639.015} C_VEL
LIN {X 0,Y 503.065,Z 333.951,A -85,B 0,C 180,E1 -5640.092,E2 -5640.092} C_VEL
LIN {X 0,Y 502.805,Z 342.041,A -85,B 0,C 180,E1 -5641.169,E2 -5641.169} C_VEL
LIN {X 0,Y 502.499,Z 350.181,A -85,B 0,C 180,E1 -5642.513,E2 -5642.513} C_VEL
LIN {X 0,Y 502.369,Z 355.213,A -85,B 0,C 180,E1 -5643.551,E2 -5643.551} C_VEL
LIN {X 0,Y 502.239,Z 359.859,A -85,B 0,C 180,E1 -5644.736,E2 -5644.736} C_VEL
LIN {X 0,Y 502.134,Z 363.797,A -85,B 0,C 180,E1 -5646.053,E2 -5646.053} C_VEL
LIN {X 0,Y 502.042,Z 366.769,A -85,B 0,C 180,E1 -5647.505,E2 -5647.505} C_VEL
LIN {X 0,Y 502.004,Z 368.144,A -85,B 0,C 180,E1 -5648.654,E2 -5648.654} C_VEL
LIN {X 0,Y 502.037,Z 368.679,A -85,B 0,C 180,E1 -5649.705,E2 -5649.705} C_VEL
LIN {X 0,Y 502.006,Z 368.301,A -85,B 0,C 180,E1 -5651.216,E2 -5651.216} C_VEL
LIN {X 0,Y 502.048,Z 367.343,A -85,B 0,C 180,E1 -5652.157,E2 -5652.157} C_VEL
LIN {X 0,Y 502.119,Z 364.476,A -85,B 0,C 180,E1 -5653.744,E2 -5653.744} C_VEL
LIN {X 0,Y 502.263,Z 361.308,A -85,B 0,C 180,E1 -5654.902,E2 -5654.902} C_VEL
LIN {X 0,Y 502.334,Z 356.456,A -85,B 0,C 180,E1 -5656.241,E2 -5656.241} C_VEL
LIN {X 0,Y 502.541,Z 349.502,A -85,B 0,C 180,E1 -5657.686,E2 -5657.686} C_VEL
LIN {X 0,Y 502.789,Z 341.957,A -85,B 0,C 180,E1 -5658.919,E2 -5658.919} C_VEL
LIN {X 0,Y 503.015,Z 334.279,A -85,B 0,C 180,E1 -5659.942,E2 -5659.942} C_VEL
LIN {X 0,Y 503.35,Z 324.941,A -85,B 0,C 180,E1 -5660.963,E2 -5660.963} C_VEL
LIN {X 0,Y 503.725,Z 314.534,A -85,B 0,C 180,E1 -5661.879,E2 -5661.879} C_VEL
LIN {X 0,Y 504.143,Z 302.559,A -85,B 0,C 180,E1 -5662.719,E2 -5662.719} C_VEL
LIN {X 0,Y 504.408,Z 290.898,A -85,B 0,C 180,E1 -5663.349,E2 -5663.349} C_VEL
LIN {X 0,Y 504.651,Z 278.198,A -85,B 0,C 180,E1 -5663.854,E2 -5663.854} C_VEL
LIN {X 0,Y 504.825,Z 264.964,A -85,B 0,C 180,E1 -5664.207,E2 -5664.207} C_VEL
LIN {X 0,Y 505.364,Z 169.095,A -85,B 0,C 180,E1 -5665.601,E2 -5665.601} C_VEL
LIN {X 0,Y 503.271,Z 158.207,A -85,B 0,C 180,E1 -5665.846,E2 -5665.846} C_VEL
LIN {X 0,Y 503.577,Z 143.076,A -85,B 0,C 180,E1 -5668.801,E2 -5668.801} C_VEL
LIN {X 0,Y 503.198,Z 137.08,A -85,B 0,C 180,E1 -5670,E2 -5670} C_VEL
LIN {X 0,Y 502.913,Z 135.844,A -85,B 0,C 180,E1 -5670.3,E2 -5670.3} C_VEL
LIN {X 0,Y 503.004,Z 135.831,A -85,B 0,C 180,E1 -5672.402,E2 -5672.402} C_VEL
LIN {X 0,Y 502.887,Z 135.842,A -85,B 0,C 180,E1 -5675.614,E2 -5675.614} C_VEL
LIN {X 0,Y 502.841,Z 135.85,A -85,B 0,C 180,E1 -5678.034,E2 -5678.034} C_VEL
LIN {X 0,Y 502.832,Z 135.847,A -85,B 0,C 180,E1 -5681.284,E2 -5681.284} C_VEL
LIN {X 0,Y 502.797,Z 135.85,A -85,B 0,C 180,E1 -5684.573,E2 -5684.573} C_VEL
LIN {X 0,Y 502.774,Z 135.857,A -85,B 0,C 180,E1 -5687.91,E2 -5687.91} C_VEL
LIN {X 0,Y 502.764,Z 135.854,A -85,B 0,C 180,E1 -5690.518,E2 -5690.518} C_VEL
LIN {X 0,Y 502.752,Z 135.858,A -85,B 0,C 180,E1 -5693.043,E2 -5693.043} C_VEL
LIN {X 0,Y 502.755,Z 135.86,A -85,B 0,C 180,E1 -5695.681,E2 -5695.681} C_VEL
LIN {X 0,Y 502.756,Z 135.855,A -85,B 0,C 180,E1 -5698.378,E2 -5698.378} C_VEL
LIN {X 0,Y 502.761,Z 135.86,A -85,B 0,C 180,E1 -5701.494,E2 -5701.494} C_VEL
LIN {X 0,Y 502.771,Z 135.853,A -85,B 0,C 180,E1 -5704.439,E2 -5704.439} C_VEL
LIN {X 0,Y 502.726,Z 135.867,A -85,B 0,C 180,E1 -5707.171,E2 -5707.171} C_VEL
LIN {X 0,Y 502.738,Z 135.857,A -85,B 0,C 180,E1 -5710.021,E2 -5710.021} C_VEL
LIN {X 0,Y 502.743,Z 135.856,A -85,B 0,C 180,E1 -5712.192,E2 -5712.192} C_VEL
LIN {X 0,Y 502.777,Z 135.854,A -85,B 0,C 180,E1 -5715.472,E2 -5715.472} C_VEL
LIN {X 0,Y 502.76,Z 135.862,A -85,B 0,C 180,E1 -5718.929,E2 -5718.929} C_VEL
LIN {X 0,Y 502.76,Z 135.855,A -85,B 0,C 180,E1 -5722.044,E2 -5722.044} C_VEL
LIN {X 0,Y 502.78,Z 135.856,A -85,B 0,C 180,E1 -5725.033,E2 -5725.033} C_VEL
LIN {X 0,Y 502.757,Z 135.855,A -85,B 0,C 180,E1 -5727.914,E2 -5727.914} C_VEL
LIN {X 0,Y 502.753,Z 135.862,A -85,B 0,C 180,E1 -5730.708,E2 -5730.708} C_VEL
LIN {X 0,Y 502.772,Z 135.853,A -85,B 0,C 180,E1 -5733.461,E2 -5733.461} C_VEL
LIN {X 0,Y 502.753,Z 135.859,A -85,B 0,C 180,E1 -5736.085,E2 -5736.085} C_VEL
LIN {X 0,Y 502.757,Z 135.859,A -85,B 0,C 180,E1 -5738.688,E2 -5738.688} C_VEL
LIN {X 0,Y 502.79,Z 135.854,A -85,B 0,C 180,E1 -5741.9,E2 -5741.9} C_VEL
LIN {X 0,Y 502.824,Z 135.849,A -85,B 0,C 180,E1 -5744.672,E2 -5744.672} C_VEL
LIN {X 0,Y 502.874,Z 135.847,A -85,B 0,C 180,E1 -5748.044,E2 -5748.044} C_VEL
LIN {X 0,Y 502.84,Z 135.844,A -85,B 0,C 180,E1 -5751.157,E2 -5751.157} C_VEL
LIN {X 0,Y 502.87,Z 135.844,A -85,B 0,C 180,E1 -5753.581,E2 -5753.581} C_VEL
LIN {X 0,Y 502.832,Z 135.845,A -85,B 0,C 180,E1 -5756.796,E2 -5756.796} C_VEL
LIN {X 0,Y 502.895,Z 135.839,A -85,B 0,C 180,E1 -5758.399,E2 -5758.399} C_VEL
LIN {X 0,Y 503.007,Z 135.83,A -85,B 0,C 180,E1 -5760,E2 -5760} C_VEL
LIN {X 0,Y 503.012,Z 135.824,A -85,B 0,C 180,E1 -5762.403,E2 -5762.403} C_VEL
LIN {X 0,Y 502.891,Z 135.845,A -85,B 0,C 180,E1 -5765.614,E2 -5765.614} C_VEL
LIN {X 0,Y 502.852,Z 135.846,A -85,B 0,C 180,E1 -5768.035,E2 -5768.035} C_VEL
LIN {X 0,Y 502.881,Z 135.844,A -85,B 0,C 180,E1 -5771.283,E2 -5771.283} C_VEL
LIN {X 0,Y 502.827,Z 135.846,A -85,B 0,C 180,E1 -5774.572,E2 -5774.572} C_VEL
LIN {X 0,Y 502.791,Z 135.852,A -85,B 0,C 180,E1 -5777.91,E2 -5777.91} C_VEL
LIN {X 0,Y 502.808,Z 135.849,A -85,B 0,C 180,E1 -5780.528,E2 -5780.528} C_VEL
LIN {X 0,Y 502.787,Z 135.856,A -85,B 0,C 180,E1 -5783.041,E2 -5783.041} C_VEL
LIN {X 0,Y 502.781,Z 135.854,A -85,B 0,C 180,E1 -5785.679,E2 -5785.679} C_VEL
LIN {X 0,Y 502.774,Z 135.853,A -85,B 0,C 180,E1 -5788.377,E2 -5788.377} C_VEL
LIN {X 0,Y 502.77,Z 135.86,A -85,B 0,C 180,E1 -5791.145,E2 -5791.145} C_VEL
LIN {X 0,Y 502.791,Z 135.85,A -85,B 0,C 180,E1 -5793.995,E2 -5793.995} C_VEL
LIN {X 0,Y 502.769,Z 135.858,A -85,B 0,C 180,E1 -5797.176,E2 -5797.176} C_VEL
LIN {X 0,Y 502.775,Z 135.853,A -85,B 0,C 180,E1 -5800.017,E2 -5800.017} C_VEL
LIN {X 0,Y 502.751,Z 135.858,A -85,B 0,C 180,E1 -5803.234,E2 -5803.234} C_VEL
LIN {X 0,Y 502.782,Z 135.851,A -85,B 0,C 180,E1 -5805.66,E2 -5805.66} C_VEL
LIN {X 0,Y 502.769,Z 135.856,A -85,B 0,C 180,E1 -5809.012,E2 -5809.012} C_VEL
LIN {X 0,Y 502.793,Z 135.852,A -85,B 0,C 180,E1 -5812.045,E2 -5812.045} C_VEL
LIN {X 0,Y 502.795,Z 135.851,A -85,B 0,C 180,E1 -5815.033,E2 -5815.033} C_VEL
LIN {X 0,Y 502.786,Z 135.853,A -85,B 0,C 180,E1 -5817.915,E2 -5817.915} C_VEL
LIN {X 0,Y 502.808,Z 135.854,A -85,B 0,C 180,E1 -5820.711,E2 -5820.711} C_VEL
LIN {X 0,Y 502.778,Z 135.857,A -85,B 0,C 180,E1 -5823.46,E2 -5823.46} C_VEL
LIN {X 0,Y 502.82,Z 136.061,A -85,B 0,C 180,E1 -5824.988,E2 -5824.988} C_VEL
LIN {X 0,Y 504.471,Z 145.113,A -85,B 0,C 180,E1 -5826.56,E2 -5826.56} C_VEL
LIN {X 0,Y 504.21,Z 157.227,A -85,B 0,C 180,E1 -5828.537,E2 -5828.537} C_VEL
LIN {X 0,Y 503.575,Z 178.275,A -85,B 0,C 180,E1 -5831.922,E2 -5831.922} C_VEL
LIN {X 0,Y 503.221,Z 192.602,A -85,B 0,C 180,E1 -5834.198,E2 -5834.198} C_VEL
LIN {X 0,Y 505.299,Z 207.908,A -85,B 0,C 180,E1 -5834.486,E2 -5834.486} C_VEL
LIN {X 0,Y 504.811,Z 301.403,A -85,B 0,C 180,E1 -5835.847,E2 -5835.847} C_VEL
LIN {X 0,Y 504.556,Z 314.536,A -85,B 0,C 180,E1 -5836.2,E2 -5836.2} C_VEL
LIN {X 0,Y 504.189,Z 327.202,A -85,B 0,C 180,E1 -5836.703,E2 -5836.703} C_VEL
LIN {X 0,Y 503.856,Z 338.318,A -85,B 0,C 180,E1 -5837.3,E2 -5837.3} C_VEL
LIN {X 0,Y 503.516,Z 350.132,A -85,B 0,C 180,E1 -5838.119,E2 -5838.119} C_VEL
LIN {X 0,Y 503.203,Z 360.631,A -85,B 0,C 180,E1 -5839.03,E2 -5839.03} C_VEL
LIN {X 0,Y 502.834,Z 369.205,A -85,B 0,C 180,E1 -5839.938,E2 -5839.938} C_VEL
LIN {X 0,Y 502.605,Z 377.116,A -85,B 0,C 180,E1 -5840.949,E2 -5840.949} C_VEL
LIN {X 0,Y 502.38,Z 384.843,A -85,B 0,C 180,E1 -5842.16,E2 -5842.16} C_VEL
LIN {X 0,Y 502.237,Z 391.552,A -85,B 0,C 180,E1 -5843.482,E2 -5843.482} C_VEL
LIN {X 0,Y 502.171,Z 396.698,A -85,B 0,C 180,E1 -5844.78,E2 -5844.78} C_VEL
LIN {X 0,Y 502.138,Z 400.317,A -85,B 0,C 180,E1 -5845.987,E2 -5845.987} C_VEL
LIN {X 0,Y 502.12,Z 402.184,A -85,B 0,C 180,E1 -5846.79,E2 -5846.79} C_VEL
LIN {X 0,Y 502.092,Z 403.582,A -85,B 0,C 180,E1 -5847.593,E2 -5847.593} C_VEL
LIN {X 0,Y 501.996,Z 405.183,A -85,B 0,C 180,E1 -5849.198,E2 -5849.198} C_VEL
LIN {X 0,Y 501.989,Z 405.398,A -85,B 0,C 180,E1 -5850,E2 -5850} C_VEL
LIN {X 0,Y 502.036,Z 404.568,A -85,B 0,C 180,E1 -5851.604,E2 -5851.604} C_VEL
LIN {X 0,Y 502.092,Z 403.568,A -85,B 0,C 180,E1 -5852.407,E2 -5852.407} C_VEL
LIN {X 0,Y 502.12,Z 402.165,A -85,B 0,C 180,E1 -5853.209,E2 -5853.209} C_VEL
LIN {X 0,Y 502.1,Z 399.213,A -85,B 0,C 180,E1 -5854.415,E2 -5854.415} C_VEL
LIN {X 0,Y 502.196,Z 395.223,A -85,B 0,C 180,E1 -5855.622,E2 -5855.622} C_VEL
LIN {X 0,Y 502.291,Z 389.185,A -85,B 0,C 180,E1 -5857.012,E2 -5857.012} C_VEL
LIN {X 0,Y 502.448,Z 382.376,A -85,B 0,C 180,E1 -5858.243,E2 -5858.243} C_VEL
LIN {X 0,Y 502.692,Z 374.062,A -85,B 0,C 180,E1 -5859.455,E2 -5859.455} C_VEL
LIN {X 0,Y 502.956,Z 365.542,A -85,B 0,C 180,E1 -5860.466,E2 -5860.466} C_VEL
LIN {X 0,Y 503.345,Z 355.023,A -85,B 0,C 180,E1 -5861.476,E2 -5861.476} C_VEL
LIN {X 0,Y 503.682,Z 343.243,A -85,B 0,C 180,E1 -5862.384,E2 -5862.384} C_VEL
LIN {X 0,Y 504.082,Z 331.279,A -85,B 0,C 180,E1 -5863.095,E2 -5863.095} C_VEL
LIN {X 0,Y 504.442,Z 318.899,A -85,B 0,C 180,E1 -5863.649,E2 -5863.649} C_VEL
LIN {X 0,Y 504.726,Z 306.183,A -85,B 0,C 180,E1 -5864.052,E2 -5864.052} C_VEL
LIN {X 0,Y 504.978,Z 291.064,A -85,B 0,C 180,E1 -5864.328,E2 -5864.328} C_VEL
LIN {X 0,Y 505.224,Z 205.884,A -85,B 0,C 180,E1 -5865.557,E2 -5865.557} C_VEL
LIN {X 0,Y 503.227,Z 192.275,A -85,B 0,C 180,E1 -5865.839,E2 -5865.839} C_VEL
LIN {X 0,Y 503.737,Z 172.83,A -85,B 0,C 180,E1 -5868.928,E2 -5868.928} C_VEL
LIN {X 0,Y 504.173,Z 155.76,A -85,B 0,C 180,E1 -5871.679,E2 -5871.679} C_VEL
LIN {X 0,Y 504.466,Z 145.029,A -85,B 0,C 180,E1 -5873.435,E2 -5873.435} C_VEL
LIN {X 0,Y 502.781,Z 135.858,A -85,B 0,C 180,E1 -5875.069,E2 -5875.069} C_VEL
LIN {X 0,Y 502.78,Z 135.86,A -85,B 0,C 180,E1 -5877.47,E2 -5877.47} C_VEL
LIN {X 0,Y 502.805,Z 135.854,A -85,B 0,C 180,E1 -5880.212,E2 -5880.212} C_VEL
LIN {X 0,Y 502.805,Z 135.853,A -85,B 0,C 180,E1 -5883.033,E2 -5883.033} C_VEL
LIN {X 0,Y 502.765,Z 135.857,A -85,B 0,C 180,E1 -5885.952,E2 -5885.952} C_VEL
LIN {X 0,Y 502.786,Z 135.857,A -85,B 0,C 180,E1 -5888.978,E2 -5888.978} C_VEL
LIN {X 0,Y 502.747,Z 135.857,A -85,B 0,C 180,E1 -5892.192,E2 -5892.192} C_VEL
LIN {X 0,Y 502.78,Z 135.856,A -85,B 0,C 180,E1 -5895.471,E2 -5895.471} C_VEL
LIN {X 0,Y 502.76,Z 135.861,A -85,B 0,C 180,E1 -5898.928,E2 -5898.928} C_VEL
LIN {X 0,Y 502.749,Z 135.855,A -85,B 0,C 180,E1 -5902.042,E2 -5902.042} C_VEL
LIN {X 0,Y 502.752,Z 135.858,A -85,B 0,C 180,E1 -5905.03,E2 -5905.03} C_VEL
LIN {X 0,Y 502.758,Z 135.855,A -85,B 0,C 180,E1 -5907.913,E2 -5907.913} C_VEL
LIN {X 0,Y 502.754,Z 135.862,A -85,B 0,C 180,E1 -5910.707,E2 -5910.707} C_VEL
LIN {X 0,Y 502.773,Z 135.85,A -85,B 0,C 180,E1 -5913.461,E2 -5913.461} C_VEL
LIN {X 0,Y 502.754,Z 135.859,A -85,B 0,C 180,E1 -5916.084,E2 -5916.084} C_VEL
LIN {X 0,Y 502.758,Z 135.859,A -85,B 0,C 180,E1 -5918.687,E2 -5918.687} C_VEL
LIN {X 0,Y 502.79,Z 135.853,A -85,B 0,C 180,E1 -5921.899,E2 -5921.899} C_VEL
LIN {X 0,Y 502.838,Z 135.847,A -85,B 0,C 180,E1 -5924.665,E2 -5924.665} C_VEL
LIN {X 0,Y 502.873,Z 135.845,A -85,B 0,C 180,E1 -5928.043,E2 -5928.043} C_VEL
LIN {X 0,Y 502.85,Z 135.842,A -85,B 0,C 180,E1 -5931.156,E2 -5931.156} C_VEL
LIN {X 0,Y 502.874,Z 135.843,A -85,B 0,C 180,E1 -5933.58,E2 -5933.58} C_VEL
LIN {X 0,Y 502.837,Z 135.84,A -85,B 0,C 180,E1 -5936.795,E2 -5936.795} C_VEL
LIN {X 0,Y 502.896,Z 135.838,A -85,B 0,C 180,E1 -5938.398,E2 -5938.398} C_VEL
LIN {X 0,Y 503.009,Z 135.825,A -85,B 0,C 180,E1 -5940,E2 -5940} C_VEL
LIN {X 0,Y 503.02,Z 135.821,A -85,B 0,C 180,E1 -5942.402,E2 -5942.402} C_VEL
LIN {X 0,Y 502.919,Z 135.838,A -85,B 0,C 180,E1 -5945.613,E2 -5945.613} C_VEL
LIN {X 0,Y 502.865,Z 135.844,A -85,B 0,C 180,E1 -5948.843,E2 -5948.843} C_VEL
LIN {X 0,Y 502.847,Z 135.844,A -85,B 0,C 180,E1 -5952.101,E2 -5952.101} C_VEL
LIN {X 0,Y 502.851,Z 135.849,A -85,B 0,C 180,E1 -5955.399,E2 -5955.399} C_VEL
LIN {X 0,Y 502.824,Z 135.85,A -85,B 0,C 180,E1 -5958.751,E2 -5958.751} C_VEL
LIN {X 0,Y 502.784,Z 135.853,A -85,B 0,C 180,E1 -5961.311,E2 -5961.311} C_VEL
LIN {X 0,Y 502.77,Z 135.855,A -85,B 0,C 180,E1 -5963.914,E2 -5963.914} C_VEL
LIN {X 0,Y 502.837,Z 135.851,A -85,B 0,C 180,E1 -5966.567,E2 -5966.567} C_VEL
LIN {X 0,Y 502.823,Z 135.849,A -85,B 0,C 180,E1 -5969.287,E2 -5969.287} C_VEL
LIN {X 0,Y 502.782,Z 135.855,A -85,B 0,C 180,E1 -5972.084,E2 -5972.084} C_VEL
LIN {X 0,Y 502.795,Z 135.855,A -85,B 0,C 180,E1 -5974.966,E2 -5974.966} C_VEL
LIN {X 0,Y 502.792,Z 135.856,A -85,B 0,C 180,E1 -5977.953,E2 -5977.953} C_VEL
LIN {X 0,Y 502.819,Z 135.851,A -85,B 0,C 180,E1 -5981.065,E2 -5981.065} C_VEL
LIN {X 0,Y 502.8,Z 135.857,A -85,B 0,C 180,E1 -5984.531,E2 -5984.531} C_VEL
LIN {X 0,Y 502.797,Z 135.858,A -85,B 0,C 180,E1 -5987.861,E2 -5987.861} C_VEL
LIN {X 0,Y 502.847,Z 135.876,A -85,B 0,C 180,E1 -5989.859,E2 -5989.859} C_VEL
LIN {X 0,Y 503.633,Z 140.973,A -85,B 0,C 180,E1 -5990.888,E2 -5990.888} C_VEL
LIN {X 0,Y 503.408,Z 155.056,A -85,B 0,C 180,E1 -5993.606,E2 -5993.606} C_VEL
LIN {X 0,Y 503.328,Z 157.735,A -85,B 0,C 180,E1 -5994.122,E2 -5994.122} C_VEL
LIN {X 0,Y 502.905,Z 159.096,A -85,B 0,C 180,E1 -5994.223,E2 -5994.223} C_VEL
LIN {X 0,Y 499.465,Z 167.504,A -85,B 0,C 180,E1 -5994.25,E2 -5994.25} C_VEL
LIN {X 0,Y 498.13,Z 173.595,A -85,B 0,C 180,E1 -5994.269,E2 -5994.269} C_VEL
LIN {X 0,Y 498.155,Z 180.158,A -85,B 0,C 180,E1 -5994.359,E2 -5994.359} C_VEL
LIN {X 0,Y 498.577,Z 188.954,A -85,B 0,C 180,E1 -5994.538,E2 -5994.538} C_VEL
LIN {X 0,Y 498.067,Z 265.303,A -85,B 0,C 180,E1 -5995.667,E2 -5995.667} C_VEL
LIN {X 0,Y 497.865,Z 277.854,A -85,B 0,C 180,E1 -5996.001,E2 -5996.001} C_VEL
LIN {X 0,Y 497.599,Z 289.992,A -85,B 0,C 180,E1 -5996.48,E2 -5996.48} C_VEL
LIN {X 0,Y 497.28,Z 300.585,A -85,B 0,C 180,E1 -5997.036,E2 -5997.036} C_VEL
LIN {X 0,Y 496.932,Z 311.324,A -85,B 0,C 180,E1 -5997.751,E2 -5997.751} C_VEL
LIN {X 0,Y 496.523,Z 322.13,A -85,B 0,C 180,E1 -5998.656,E2 -5998.656} C_VEL
LIN {X 0,Y 496.15,Z 332.764,A -85,B 0,C 180,E1 -5999.775,E2 -5999.775} C_VEL
LIN {X 0,Y 495.799,Z 341.759,A -85,B 0,C 180,E1 -6000.955,E2 -6000.955} C_VEL
LIN {X 0,Y 495.51,Z 348.769,A -85,B 0,C 180,E1 -6002.092,E2 -6002.092} C_VEL
LIN {X 0,Y 495.351,Z 355.054,A -85,B 0,C 180,E1 -6003.358,E2 -6003.358} C_VEL
LIN {X 0,Y 495.163,Z 360.618,A -85,B 0,C 180,E1 -6004.799,E2 -6004.799} C_VEL
LIN {X 0,Y 495.048,Z 364.423,A -85,B 0,C 180,E1 -6006.134,E2 -6006.134} C_VEL
LIN {X 0,Y 494.957,Z 367.019,A -85,B 0,C 180,E1 -6007.457,E2 -6007.457} C_VEL
LIN {X 0,Y 494.91,Z 368.116,A -85,B 0,C 180,E1 -6008.333,E2 -6008.333} C_VEL
LIN {X 0,Y 494.946,Z 368.916,A -85,B 0,C 180,E1 -6009.58,E2 -6009.58} C_VEL
LIN {X 0,Y 494.934,Z 368.731,A -85,B 0,C 180,E1 -6010.938,E2 -6010.938} C_VEL
LIN {X 0,Y 494.944,Z 367.775,A -85,B 0,C 180,E1 -6012.057,E2 -6012.057} C_VEL
LIN {X 0,Y 495.023,Z 365.361,A -85,B 0,C 180,E1 -6013.504,E2 -6013.504} C_VEL
LIN {X 0,Y 495.187,Z 362.021,A -85,B 0,C 180,E1 -6014.816,E2 -6014.816} C_VEL
LIN {X 0,Y 495.243,Z 357.826,A -85,B 0,C 180,E1 -6016.04,E2 -6016.04} C_VEL
LIN {X 0,Y 495.464,Z 351.261,A -85,B 0,C 180,E1 -6017.507,E2 -6017.507} C_VEL
LIN {X 0,Y 495.694,Z 344.063,A -85,B 0,C 180,E1 -6018.758,E2 -6018.758} C_VEL
LIN {X 0,Y 495.988,Z 335.106,A -85,B 0,C 180,E1 -6020.004,E2 -6020.004} C_VEL
LIN {X 0,Y 496.344,Z 325.91,A -85,B 0,C 180,E1 -6021.04,E2 -6021.04} C_VEL
LIN {X 0,Y 496.774,Z 315.124,A -85,B 0,C 180,E1 -6022.013,E2 -6022.013} C_VEL
LIN {X 0,Y 497.148,Z 304.338,A -85,B 0,C 180,E1 -6022.793,E2 -6022.793} C_VEL
LIN {X 0,Y 497.463,Z 292.619,A -85,B 0,C 180,E1 -6023.46,E2 -6023.46} C_VEL
LIN {X 0,Y 497.73,Z 279.79,A -85,B 0,C 180,E1 -6023.997,E2 -6023.997} C_VEL
LIN {X 0,Y 497.958,Z 267.143,A -85,B 0,C 180,E1 -6024.356,E2 -6024.356} C_VEL
LIN {X 0,Y 498.138,Z 239.531,A -85,B 0,C 180,E1 -6024.789,E2 -6024.789} C_VEL
LIN {X 0,Y 498.534,Z 169.878,A -85,B 0,C 180,E1 -6025.806,E2 -6025.806} C_VEL
LIN {X 0,Y 496.31,Z 158.426,A -85,B 0,C 180,E1 -6026.067,E2 -6026.067} C_VEL
LIN {X 0,Y 496.598,Z 143.62,A -85,B 0,C 180,E1 -6028.987,E2 -6028.987} C_VEL
LIN {X 0,Y 496.039,Z 137.625,A -85,B 0,C 180,E1 -6030.203,E2 -6030.203} C_VEL
LIN {X 0,Y 495.816,Z 136.727,A -85,B 0,C 180,E1 -6030.406,E2 -6030.406} C_VEL
LIN {X 0,Y 495.97,Z 136.707,A -85,B 0,C 180,E1 -6032.437,E2 -6032.437} C_VEL
LIN {X 0,Y 495.845,Z 136.721,A -85,B 0,C 180,E1 -6035.694,E2 -6035.694} C_VEL
LIN {X 0,Y 495.805,Z 136.725,A -85,B 0,C 180,E1 -6038.149,E2 -6038.149} C_VEL
LIN {X 0,Y 495.817,Z 136.723,A -85,B 0,C 180,E1 -6041.446,E2 -6041.446} C_VEL
LIN {X 0,Y 495.751,Z 136.727,A -85,B 0,C 180,E1 -6044.784,E2 -6044.784} C_VEL
LIN {X 0,Y 495.743,Z 136.73,A -85,B 0,C 180,E1 -6048.226,E2 -6048.226} C_VEL
LIN {X 0,Y 495.718,Z 136.739,A -85,B 0,C 180,E1 -6051.63,E2 -6051.63} C_VEL
LIN {X 0,Y 495.692,Z 136.735,A -85,B 0,C 180,E1 -6054.278,E2 -6054.278} C_VEL
LIN {X 0,Y 495.713,Z 136.735,A -85,B 0,C 180,E1 -6056.98,E2 -6056.98} C_VEL
LIN {X 0,Y 495.691,Z 136.738,A -85,B 0,C 180,E1 -6059.752,E2 -6059.752} C_VEL
LIN {X 0,Y 495.721,Z 136.732,A -85,B 0,C 180,E1 -6062.598,E2 -6062.598} C_VEL
LIN {X 0,Y 495.723,Z 136.735,A -85,B 0,C 180,E1 -6065.54,E2 -6065.54} C_VEL
LIN {X 0,Y 495.73,Z 136.734,A -85,B 0,C 180,E1 -6068.764,E2 -6068.764} C_VEL
LIN {X 0,Y 495.72,Z 136.732,A -85,B 0,C 180,E1 -6071.785,E2 -6071.785} C_VEL
LIN {X 0,Y 495.73,Z 136.736,A -85,B 0,C 180,E1 -6075.142,E2 -6075.142} C_VEL
LIN {X 0,Y 495.722,Z 136.732,A -85,B 0,C 180,E1 -6078.216,E2 -6078.216} C_VEL
LIN {X 0,Y 495.737,Z 136.732,A -85,B 0,C 180,E1 -6081.236,E2 -6081.236} C_VEL
LIN {X 0,Y 495.728,Z 136.735,A -85,B 0,C 180,E1 -6084.461,E2 -6084.461} C_VEL
LIN {X 0,Y 495.725,Z 136.731,A -85,B 0,C 180,E1 -6087.403,E2 -6087.403} C_VEL
LIN {X 0,Y 495.696,Z 136.738,A -85,B 0,C 180,E1 -6090.25,E2 -6090.25} C_VEL
LIN {X 0,Y 495.722,Z 136.731,A -85,B 0,C 180,E1 -6093.275,E2 -6093.275} C_VEL
LIN {X 0,Y 495.703,Z 136.734,A -85,B 0,C 180,E1 -6095.723,E2 -6095.723} C_VEL
LIN {X 0,Y 495.725,Z 136.739,A -85,B 0,C 180,E1 -6098.371,E2 -6098.371} C_VEL
LIN {X 0,Y 495.75,Z 136.729,A -85,B 0,C 180,E1 -6101.775,E2 -6101.775} C_VEL
LIN {X 0,Y 495.757,Z 136.727,A -85,B 0,C 180,E1 -6105.217,E2 -6105.217} C_VEL
LIN {X 0,Y 495.825,Z 136.721,A -85,B 0,C 180,E1 -6108.555,E2 -6108.555} C_VEL
LIN {X 0,Y 495.814,Z 136.725,A -85,B 0,C 180,E1 -6111.852,E2 -6111.852} C_VEL
LIN {X 0,Y 495.853,Z 136.719,A -85,B 0,C 180,E1 -6114.306,E2 -6114.306} C_VEL
LIN {X 0,Y 495.979,Z 136.703,A -85,B 0,C 180,E1 -6117.564,E2 -6117.564} C_VEL
LIN {X 0,Y 495.976,Z 136.705,A -85,B 0,C 180,E1 -6120,E2 -6120} C_VEL
LIN {X 0,Y 495.978,Z 136.7,A -85,B 0,C 180,E1 -6122.437,E2 -6122.437} C_VEL
LIN {X 0,Y 495.849,Z 136.724,A -85,B 0,C 180,E1 -6125.694,E2 -6125.694} C_VEL
LIN {X 0,Y 495.816,Z 136.721,A -85,B 0,C 180,E1 -6128.149,E2 -6128.149} C_VEL
LIN {X 0,Y 495.856,Z 136.721,A -85,B 0,C 180,E1 -6131.445,E2 -6131.445} C_VEL
LIN {X 0,Y 495.779,Z 136.725,A -85,B 0,C 180,E1 -6134.784,E2 -6134.784} C_VEL
LIN {X 0,Y 495.778,Z 136.724,A -85,B 0,C 180,E1 -6138.235,E2 -6138.235} C_VEL
LIN {X 0,Y 495.769,Z 136.727,A -85,B 0,C 180,E1 -6140.757,E2 -6140.757} C_VEL
LIN {X 0,Y 495.739,Z 136.735,A -85,B 0,C 180,E1 -6143.388,E2 -6143.388} C_VEL
LIN {X 0,Y 495.721,Z 136.731,A -85,B 0,C 180,E1 -6146.072,E2 -6146.072} C_VEL
LIN {X 0,Y 495.723,Z 136.735,A -85,B 0,C 180,E1 -6148.818,E2 -6148.818} C_VEL
LIN {X 0,Y 495.742,Z 136.729,A -85,B 0,C 180,E1 -6151.722,E2 -6151.722} C_VEL
LIN {X 0,Y 495.764,Z 136.73,A -85,B 0,C 180,E1 -6154.692,E2 -6154.692} C_VEL
LIN {X 0,Y 495.725,Z 136.731,A -85,B 0,C 180,E1 -6157.562,E2 -6157.562} C_VEL
LIN {X 0,Y 495.748,Z 136.728,A -85,B 0,C 180,E1 -6160.045,E2 -6160.045} C_VEL
LIN {X 0,Y 495.699,Z 136.741,A -85,B 0,C 180,E1 -6162.886,E2 -6162.886} C_VEL
LIN {X 0,Y 495.726,Z 136.731,A -85,B 0,C 180,E1 -6165.998,E2 -6165.998} C_VEL
LIN {X 0,Y 495.732,Z 136.731,A -85,B 0,C 180,E1 -6169.296,E2 -6169.296} C_VEL
LIN {X 0,Y 495.749,Z 136.728,A -85,B 0,C 180,E1 -6171.408,E2 -6171.408} C_VEL
LIN {X 0,Y 495.747,Z 136.737,A -85,B 0,C 180,E1 -6174.462,E2 -6174.462} C_VEL
LIN {X 0,Y 495.756,Z 136.727,A -85,B 0,C 180,E1 -6177.404,E2 -6177.404} C_VEL
LIN {X 0,Y 495.761,Z 136.734,A -85,B 0,C 180,E1 -6180.253,E2 -6180.253} C_VEL
LIN {X 0,Y 495.743,Z 136.733,A -85,B 0,C 180,E1 -6183.27,E2 -6183.27} C_VEL
LIN {X 0,Y 495.76,Z 136.874,A -85,B 0,C 180,E1 -6184.803,E2 -6184.803} C_VEL
LIN {X 0,Y 497.529,Z 146.512,A -85,B 0,C 180,E1 -6186.503,E2 -6186.503} C_VEL
LIN {X 0,Y 497.165,Z 161.832,A -85,B 0,C 180,E1 -6189.029,E2 -6189.029} C_VEL
LIN {X 0,Y 496.505,Z 181.84,A -85,B 0,C 180,E1 -6192.282,E2 -6192.282} C_VEL
LIN {X 0,Y 496.223,Z 192.278,A -85,B 0,C 180,E1 -6193.964,E2 -6193.964} C_VEL
LIN {X 0,Y 498.436,Z 207.55,A -85,B 0,C 180,E1 -6194.27,E2 -6194.27} C_VEL
LIN {X 0,Y 497.931,Z 300.848,A -85,B 0,C 180,E1 -6195.647,E2 -6195.647} C_VEL
LIN {X 0,Y 497.665,Z 314.078,A -85,B 0,C 180,E1 -6196.005,E2 -6196.005} C_VEL
LIN {X 0,Y 497.265,Z 326.795,A -85,B 0,C 180,E1 -6196.514,E2 -6196.514} C_VEL
LIN {X 0,Y 496.895,Z 337.95,A -85,B 0,C 180,E1 -6197.119,E2 -6197.119} C_VEL
LIN {X 0,Y 496.489,Z 349.787,A -85,B 0,C 180,E1 -6197.948,E2 -6197.948} C_VEL
LIN {X 0,Y 496.184,Z 360.302,A -85,B 0,C 180,E1 -6198.873,E2 -6198.873} C_VEL
LIN {X 0,Y 495.811,Z 368.893,A -85,B 0,C 180,E1 -6199.794,E2 -6199.794} C_VEL
LIN {X 0,Y 495.539,Z 376.82,A -85,B 0,C 180,E1 -6200.819,E2 -6200.819} C_VEL
LIN {X 0,Y 495.319,Z 384.563,A -85,B 0,C 180,E1 -6202.048,E2 -6202.048} C_VEL
LIN {X 0,Y 495.172,Z 389.861,A -85,B 0,C 180,E1 -6203.071,E2 -6203.071} C_VEL
LIN {X 0,Y 495.112,Z 394.998,A -85,B 0,C 180,E1 -6204.297,E2 -6204.297} C_VEL
LIN {X 0,Y 495.006,Z 398.981,A -85,B 0,C 180,E1 -6205.521,E2 -6205.521} C_VEL
LIN {X 0,Y 495.042,Z 401.924,A -85,B 0,C 180,E1 -6206.744,E2 -6206.744} C_VEL
LIN {X 0,Y 494.999,Z 403.323,A -85,B 0,C 180,E1 -6207.559,E2 -6207.559} C_VEL
LIN {X 0,Y 494.963,Z 404.319,A -85,B 0,C 180,E1 -6208.373,E2 -6208.373} C_VEL
LIN {X 0,Y 494.907,Z 405.139,A -85,B 0,C 180,E1 -6210,E2 -6210} C_VEL
LIN {X 0,Y 494.963,Z 404.309,A -85,B 0,C 180,E1 -6211.627,E2 -6211.627} C_VEL
LIN {X 0,Y 494.998,Z 403.308,A -85,B 0,C 180,E1 -6212.441,E2 -6212.441} C_VEL
LIN {X 0,Y 495.042,Z 401.906,A -85,B 0,C 180,E1 -6213.255,E2 -6213.255} C_VEL
LIN {X 0,Y 495.006,Z 398.954,A -85,B 0,C 180,E1 -6214.479,E2 -6214.479} C_VEL
LIN {X 0,Y 495.11,Z 394.965,A -85,B 0,C 180,E1 -6215.702,E2 -6215.702} C_VEL
LIN {X 0,Y 495.24,Z 388.832,A -85,B 0,C 180,E1 -6217.133,E2 -6217.133} C_VEL
LIN {X 0,Y 495.405,Z 382.133,A -85,B 0,C 180,E1 -6218.361,E2 -6218.361} C_VEL
LIN {X 0,Y 495.652,Z 373.825,A -85,B 0,C 180,E1 -6219.591,E2 -6219.591} C_VEL
LIN {X 0,Y 495.959,Z 365.313,A -85,B 0,C 180,E1 -6220.615,E2 -6220.615} C_VEL
LIN {X 0,Y 496.359,Z 354.801,A -85,B 0,C 180,E1 -6221.64,E2 -6221.64} C_VEL
LIN {X 0,Y 496.73,Z 343.193,A -85,B 0,C 180,E1 -6222.548,E2 -6222.548} C_VEL
LIN {X 0,Y 497.14,Z 331.086,A -85,B 0,C 180,E1 -6223.281,E2 -6223.281} C_VEL
LIN {X 0,Y 497.554,Z 318.731,A -85,B 0,C 180,E1 -6223.842,E2 -6223.842} C_VEL
LIN {X 0,Y 497.843,Z 306.061,A -85,B 0,C 180,E1 -6224.251,E2 -6224.251} C_VEL
LIN {X 0,Y 498.107,Z 292.855,A -85,B 0,C 180,E1 -6224.504,E2 -6224.504} C_VEL
LIN {X 0,Y 498.332,Z 206.131,A -85,B 0,C 180,E1 -6225.775,E2 -6225.775} C_VEL
LIN {X 0,Y 496.216,Z 191.997,A -85,B 0,C 180,E1 -6226.075,E2 -6226.075} C_VEL
LIN {X 0,Y 496.735,Z 173.905,A -85,B 0,C 180,E1 -6228.991,E2 -6228.991} C_VEL
LIN {X 0,Y 497.31,Z 155.587,A -85,B 0,C 180,E1 -6231.993,E2 -6231.993} C_VEL
LIN {X 0,Y 497.537,Z 146.417,A -85,B 0,C 180,E1 -6233.518,E2 -6233.518} C_VEL
LIN {X 0,Y 495.744,Z 136.735,A -85,B 0,C 180,E1 -6235.282,E2 -6235.282} C_VEL
LIN {X 0,Y 495.739,Z 136.734,A -85,B 0,C 180,E1 -6238.482,E2 -6238.482} C_VEL
LIN {X 0,Y 495.75,Z 136.732,A -85,B 0,C 180,E1 -6240.688,E2 -6240.688} C_VEL
LIN {X 0,Y 495.743,Z 136.735,A -85,B 0,C 180,E1 -6243.566,E2 -6243.566} C_VEL
LIN {X 0,Y 495.715,Z 136.733,A -85,B 0,C 180,E1 -6246.545,E2 -6246.545} C_VEL
LIN {X 0,Y 495.744,Z 136.732,A -85,B 0,C 180,E1 -6249.639,E2 -6249.639} C_VEL
LIN {X 0,Y 495.697,Z 136.74,A -85,B 0,C 180,E1 -6252.886,E2 -6252.886} C_VEL
LIN {X 0,Y 495.715,Z 136.733,A -85,B 0,C 180,E1 -6255.996,E2 -6255.996} C_VEL
LIN {X 0,Y 495.717,Z 136.736,A -85,B 0,C 180,E1 -6259.295,E2 -6259.295} C_VEL
LIN {X 0,Y 495.713,Z 136.734,A -85,B 0,C 180,E1 -6261.405,E2 -6261.405} C_VEL
LIN {X 0,Y 495.715,Z 136.737,A -85,B 0,C 180,E1 -6264.459,E2 -6264.459} C_VEL
LIN {X 0,Y 495.726,Z 136.732,A -85,B 0,C 180,E1 -6267.402,E2 -6267.402} C_VEL
LIN {X 0,Y 495.697,Z 136.736,A -85,B 0,C 180,E1 -6270.249,E2 -6270.249} C_VEL
LIN {X 0,Y 495.723,Z 136.728,A -85,B 0,C 180,E1 -6273.275,E2 -6273.275} C_VEL
LIN {X 0,Y 495.703,Z 136.734,A -85,B 0,C 180,E1 -6275.722,E2 -6275.722} C_VEL
LIN {X 0,Y 495.726,Z 136.735,A -85,B 0,C 180,E1 -6278.37,E2 -6278.37} C_VEL
LIN {X 0,Y 495.75,Z 136.729,A -85,B 0,C 180,E1 -6281.774,E2 -6281.774} C_VEL
LIN {X 0,Y 495.779,Z 136.724,A -85,B 0,C 180,E1 -6285.216,E2 -6285.216} C_VEL
LIN {X 0,Y 495.825,Z 136.72,A -85,B 0,C 180,E1 -6288.554,E2 -6288.554} C_VEL
LIN {X 0,Y 495.816,Z 136.722,A -85,B 0,C 180,E1 -6291.851,E2 -6291.851} C_VEL
LIN {X 0,Y 495.858,Z 136.716,A -85,B 0,C 180,E1 -6294.306,E2 -6294.306} C_VEL
LIN {X 0,Y 495.98,Z 136.7,A -85,B 0,C 180,E1 -6297.563,E2 -6297.563} C_VEL
LIN {X 0,Y 495.978,Z 136.701,A -85,B 0,C 180,E1 -6300,E2 -6300} C_VEL
LIN {X 0,Y 495.988,Z 136.697,A -85,B 0,C 180,E1 -6302.436,E2 -6302.436} C_VEL
LIN {X 0,Y 495.874,Z 136.714,A -85,B 0,C 180,E1 -6305.693,E2 -6305.693} C_VEL
LIN {X 0,Y 495.835,Z 136.721,A -85,B 0,C 180,E1 -6308.969,E2 -6308.969} C_VEL
LIN {X 0,Y 495.831,Z 136.719,A -85,B 0,C 180,E1 -6312.034,E2 -6312.034} C_VEL
LIN {X 0,Y 495.826,Z 136.723,A -85,B 0,C 180,E1 -6315.451,E2 -6315.451} C_VEL
LIN {X 0,Y 495.78,Z 136.729,A -85,B 0,C 180,E1 -6319.028,E2 -6319.028} C_VEL
LIN {X 0,Y 495.743,Z 136.728,A -85,B 0,C 180,E1 -6321.628,E2 -6321.628} C_VEL
LIN {X 0,Y 495.717,Z 136.735,A -85,B 0,C 180,E1 -6324.276,E2 -6324.276} C_VEL
LIN {X 0,Y 495.785,Z 136.729,A -85,B 0,C 180,E1 -6326.975,E2 -6326.975} C_VEL
LIN {X 0,Y 495.766,Z 136.727,A -85,B 0,C 180,E1 -6329.746,E2 -6329.746} C_VEL
LIN {X 0,Y 495.766,Z 136.733,A -85,B 0,C 180,E1 -6332.594,E2 -6332.594} C_VEL
LIN {X 0,Y 495.746,Z 136.73,A -85,B 0,C 180,E1 -6335.537,E2 -6335.537} C_VEL
LIN {X 0,Y 495.762,Z 136.731,A -85,B 0,C 180,E1 -6338.768,E2 -6338.768} C_VEL
LIN {X 0,Y 495.756,Z 136.733,A -85,B 0,C 180,E1 -6341.78,E2 -6341.78} C_VEL
LIN {X 0,Y 495.748,Z 136.731,A -85,B 0,C 180,E1 -6345.139,E2 -6345.139} C_VEL
LIN {X 0,Y 495.759,Z 136.735,A -85,B 0,C 180,E1 -6348.219,E2 -6348.219} C_VEL
LIN {X 0,Y 495.82,Z 136.845,A -85,B 0,C 180,E1 -6349.718,E2 -6349.718} C_VEL
LIN {X 0,Y 496.672,Z 142.219,A -85,B 0,C 180,E1 -6350.82,E2 -6350.82} C_VEL
LIN {X 0,Y 496.425,Z 156.065,A -85,B 0,C 180,E1 -6353.515,E2 -6353.515} C_VEL
LIN {X 0,Y 496.352,Z 158.637,A -85,B 0,C 180,E1 -6354.011,E2 -6354.011} C_VEL
LIN {X 0,Y 498.744,Z 171.819,A -85,B 0,C 180,E1 -6354.289,E2 -6354.289} C_VEL
LIN {X 0,Y 498.577,Z 188.954,A -85,B 0,C 180,E1 -6354.538,E2 -6354.538} C_VEL
LIN {X 0,Y 497.8,Z 194.795,A -85,B 0,C 180,E1 -6354.598,E2 -6354.598} C_VEL
LIN {X 0,Y 492.207,Z 213.797,A -85,B 0,C 180,E1 -6354.697,E2 -6354.697} C_VEL
LIN {X 0,Y 491.533,Z 219.636,A -85,B 0,C 180,E1 -6354.762,E2 -6354.762} C_VEL
LIN {X 0,Y 491.2,Z 265.78,A -85,B 0,C 180,E1 -6355.462,E2 -6355.462} C_VEL
LIN {X 0,Y 490.991,Z 278.734,A -85,B 0,C 180,E1 -6355.818,E2 -6355.818} C_VEL
LIN {X 0,Y 490.667,Z 291.712,A -85,B 0,C 180,E1 -6356.349,E2 -6356.349} C_VEL
LIN {X 0,Y 490.308,Z 303.327,A -85,B 0,C 180,E1 -6356.997,E2 -6356.997} C_VEL
LIN {X 0,Y 489.895,Z 314.774,A -85,B 0,C 180,E1 -6357.822,E2 -6357.822} C_VEL
LIN {X 0,Y 489.468,Z 325.125,A -85,B 0,C 180,E1 -6358.755,E2 -6358.755} C_VEL
LIN {X 0,Y 489.103,Z 334.557,A -85,B 0,C 180,E1 -6359.807,E2 -6359.807} C_VEL
LIN {X 0,Y 488.732,Z 343.621,A -85,B 0,C 180,E1 -6361.066,E2 -6361.066} C_VEL
LIN {X 0,Y 488.415,Z 351.051,A -85,B 0,C 180,E1 -6362.351,E2 -6362.351} C_VEL
LIN {X 0,Y 488.274,Z 356.368,A -85,B 0,C 180,E1 -6363.5,E2 -6363.5} C_VEL
LIN {X 0,Y 488.09,Z 361.172,A -85,B 0,C 180,E1 -6364.805,E2 -6364.805} C_VEL
LIN {X 0,Y 487.957,Z 365.003,A -85,B 0,C 180,E1 -6366.216,E2 -6366.216} C_VEL
LIN {X 0,Y 487.915,Z 366.917,A -85,B 0,C 180,E1 -6367.199,E2 -6367.199} C_VEL
LIN {X 0,Y 487.837,Z 368.072,A -85,B 0,C 180,E1 -6368.002,E2 -6368.002} C_VEL
LIN {X 0,Y 487.864,Z 369.153,A -85,B 0,C 180,E1 -6369.449,E2 -6369.449} C_VEL
LIN {X 0,Y 487.829,Z 369.142,A -85,B 0,C 180,E1 -6370.649,E2 -6370.649} C_VEL
LIN {X 0,Y 487.86,Z 368.182,A -85,B 0,C 180,E1 -6371.947,E2 -6371.947} C_VEL
LIN {X 0,Y 487.905,Z 366.213,A -85,B 0,C 180,E1 -6373.256,E2 -6373.256} C_VEL
LIN {X 0,Y 488.092,Z 362.708,A -85,B 0,C 180,E1 -6374.735,E2 -6374.735} C_VEL
LIN {X 0,Y 488.207,Z 357.543,A -85,B 0,C 180,E1 -6376.259,E2 -6376.259} C_VEL
LIN {X 0,Y 488.416,Z 351.872,A -85,B 0,C 180,E1 -6377.535,E2 -6377.535} C_VEL
LIN {X 0,Y 488.652,Z 344.795,A -85,B 0,C 180,E1 -6378.804,E2 -6378.804} C_VEL
LIN {X 0,Y 488.962,Z 335.932,A -85,B 0,C 180,E1 -6380.068,E2 -6380.068} C_VEL
LIN {X 0,Y 489.343,Z 326.845,A -85,B 0,C 180,E1 -6381.119,E2 -6381.119} C_VEL
LIN {X 0,Y 489.773,Z 316.598,A -85,B 0,C 180,E1 -6382.08,E2 -6382.08} C_VEL
LIN {X 0,Y 490.18,Z 305.688,A -85,B 0,C 180,E1 -6382.897,E2 -6382.897} C_VEL
LIN {X 0,Y 490.54,Z 293.254,A -85,B 0,C 180,E1 -6383.625,E2 -6383.625} C_VEL
LIN {X 0,Y 490.837,Z 280.611,A -85,B 0,C 180,E1 -6384.17,E2 -6384.17} C_VEL
LIN {X 0,Y 491.076,Z 268.246,A -85,B 0,C 180,E1 -6384.534,E2 -6384.534} C_VEL
LIN {X 0,Y 491.259,Z 248.058,A -85,B 0,C 180,E1 -6384.87,E2 -6384.87} C_VEL
LIN {X 0,Y 491.691,Z 170.653,A -85,B 0,C 180,E1 -6386.017,E2 -6386.017} C_VEL
LIN {X 0,Y 489.305,Z 158.658,A -85,B 0,C 180,E1 -6386.294,E2 -6386.294} C_VEL
LIN {X 0,Y 489.638,Z 144.158,A -85,B 0,C 180,E1 -6389.178,E2 -6389.178} C_VEL
LIN {X 0,Y 489.323,Z 140.132,A -85,B 0,C 180,E1 -6390,E2 -6390} C_VEL
LIN {X 0,Y 488.752,Z 137.607,A -85,B 0,C 180,E1 -6390.567,E2 -6390.567} C_VEL
LIN {X 0,Y 488.936,Z 137.584,A -85,B 0,C 180,E1 -6392.472,E2 -6392.472} C_VEL
LIN {X 0,Y 488.805,Z 137.599,A -85,B 0,C 180,E1 -6395.777,E2 -6395.777} C_VEL
LIN {X 0,Y 488.752,Z 137.602,A -85,B 0,C 180,E1 -6398.268,E2 -6398.268} C_VEL
LIN {X 0,Y 488.779,Z 137.602,A -85,B 0,C 180,E1 -6401.613,E2 -6401.613} C_VEL
LIN {X 0,Y 488.715,Z 137.604,A -85,B 0,C 180,E1 -6405.002,E2 -6405.002} C_VEL
LIN {X 0,Y 488.697,Z 137.606,A -85,B 0,C 180,E1 -6408.445,E2 -6408.445} C_VEL
LIN {X 0,Y 488.673,Z 137.611,A -85,B 0,C 180,E1 -6411.073,E2 -6411.073} C_VEL
LIN {X 0,Y 488.647,Z 137.617,A -85,B 0,C 180,E1 -6413.748,E2 -6413.748} C_VEL
LIN {X 0,Y 488.663,Z 137.61,A -85,B 0,C 180,E1 -6416.478,E2 -6416.478} C_VEL
LIN {X 0,Y 488.655,Z 137.619,A -85,B 0,C 180,E1 -6419.275,E2 -6419.275} C_VEL
LIN {X 0,Y 488.675,Z 137.609,A -85,B 0,C 180,E1 -6422.15,E2 -6422.15} C_VEL
LIN {X 0,Y 488.699,Z 137.613,A -85,B 0,C 180,E1 -6425.117,E2 -6425.117} C_VEL
LIN {X 0,Y 488.648,Z 137.612,A -85,B 0,C 180,E1 -6428.204,E2 -6428.204} C_VEL
LIN {X 0,Y 488.656,Z 137.615,A -85,B 0,C 180,E1 -6431.422,E2 -6431.422} C_VEL
LIN {X 0,Y 488.694,Z 137.613,A -85,B 0,C 180,E1 -6434.804,E2 -6434.804} C_VEL
LIN {X 0,Y 488.647,Z 137.614,A -85,B 0,C 180,E1 -6437.47,E2 -6437.47} C_VEL
LIN {X 0,Y 488.703,Z 137.605,A -85,B 0,C 180,E1 -6439.674,E2 -6439.674} C_VEL
LIN {X 0,Y 488.65,Z 137.619,A -85,B 0,C 180,E1 -6442.839,E2 -6442.839} C_VEL
LIN {X 0,Y 488.708,Z 137.605,A -85,B 0,C 180,E1 -6445.886,E2 -6445.886} C_VEL
LIN {X 0,Y 488.659,Z 137.616,A -85,B 0,C 180,E1 -6448.818,E2 -6448.818} C_VEL
LIN {X 0,Y 488.685,Z 137.608,A -85,B 0,C 180,E1 -6451.668,E2 -6451.668} C_VEL
LIN {X 0,Y 488.694,Z 137.609,A -85,B 0,C 180,E1 -6454.961,E2 -6454.961} C_VEL
LIN {X 0,Y 488.683,Z 137.612,A -85,B 0,C 180,E1 -6458.043,E2 -6458.043} C_VEL
LIN {X 0,Y 488.687,Z 137.611,A -85,B 0,C 180,E1 -6460.685,E2 -6460.685} C_VEL
LIN {X 0,Y 488.688,Z 137.614,A -85,B 0,C 180,E1 -6464.143,E2 -6464.143} C_VEL
LIN {X 0,Y 488.703,Z 137.607,A -85,B 0,C 180,E1 -6466.698,E2 -6466.698} C_VEL
LIN {X 0,Y 488.787,Z 137.6,A -85,B 0,C 180,E1 -6468.388,E2 -6468.388} C_VEL
LIN {X 0,Y 488.758,Z 137.603,A -85,B 0,C 180,E1 -6471.733,E2 -6471.733} C_VEL
LIN {X 0,Y 488.814,Z 137.597,A -85,B 0,C 180,E1 -6474.224,E2 -6474.224} C_VEL
LIN {X 0,Y 488.944,Z 137.579,A -85,B 0,C 180,E1 -6477.529,E2 -6477.529} C_VEL
LIN {X 0,Y 488.945,Z 137.581,A -85,B 0,C 180,E1 -6480,E2 -6480} C_VEL
LIN {X 0,Y 488.944,Z 137.576,A -85,B 0,C 180,E1 -6482.472,E2 -6482.472} C_VEL
LIN {X 0,Y 488.808,Z 137.6,A -85,B 0,C 180,E1 -6485.777,E2 -6485.777} C_VEL
LIN {X 0,Y 488.762,Z 137.599,A -85,B 0,C 180,E1 -6488.268,E2 -6488.268} C_VEL
LIN {X 0,Y 488.811,Z 137.599,A -85,B 0,C 180,E1 -6491.613,E2 -6491.613} C_VEL
LIN {X 0,Y 488.751,Z 137.602,A -85,B 0,C 180,E1 -6495.001,E2 -6495.001} C_VEL
LIN {X 0,Y 488.749,Z 137.6,A -85,B 0,C 180,E1 -6498.443,E2 -6498.443} C_VEL
LIN {X 0,Y 488.705,Z 137.61,A -85,B 0,C 180,E1 -6501.071,E2 -6501.071} C_VEL
LIN {X 0,Y 488.67,Z 137.612,A -85,B 0,C 180,E1 -6503.747,E2 -6503.747} C_VEL
LIN {X 0,Y 488.686,Z 137.608,A -85,B 0,C 180,E1 -6506.476,E2 -6506.476} C_VEL
LIN {X 0,Y 488.693,Z 137.613,A -85,B 0,C 180,E1 -6509.273,E2 -6509.273} C_VEL
LIN {X 0,Y 488.695,Z 137.606,A -85,B 0,C 180,E1 -6512.148,E2 -6512.148} C_VEL
LIN {X 0,Y 488.717,Z 137.61,A -85,B 0,C 180,E1 -6515.116,E2 -6515.116} C_VEL
LIN {X 0,Y 488.679,Z 137.609,A -85,B 0,C 180,E1 -6518.201,E2 -6518.201} C_VEL
LIN {X 0,Y 488.698,Z 137.608,A -85,B 0,C 180,E1 -6520.341,E2 -6520.341} C_VEL
LIN {X 0,Y 488.677,Z 137.609,A -85,B 0,C 180,E1 -6523.656,E2 -6523.656} C_VEL
LIN {X 0,Y 488.678,Z 137.612,A -85,B 0,C 180,E1 -6526.344,E2 -6526.344} C_VEL
LIN {X 0,Y 488.708,Z 137.605,A -85,B 0,C 180,E1 -6529.673,E2 -6529.673} C_VEL
LIN {X 0,Y 488.674,Z 137.613,A -85,B 0,C 180,E1 -6532.84,E2 -6532.84} C_VEL
LIN {X 0,Y 488.722,Z 137.605,A -85,B 0,C 180,E1 -6535.886,E2 -6535.886} C_VEL
LIN {X 0,Y 488.693,Z 137.611,A -85,B 0,C 180,E1 -6538.82,E2 -6538.82} C_VEL
LIN {X 0,Y 488.698,Z 137.609,A -85,B 0,C 180,E1 -6541.668,E2 -6541.668} C_VEL
LIN {X 0,Y 488.72,Z 137.699,A -85,B 0,C 180,E1 -6544.616,E2 -6544.616} C_VEL
LIN {X 0,Y 490.607,Z 148.026,A -85,B 0,C 180,E1 -6546.464,E2 -6546.464} C_VEL
LIN {X 0,Y 490.179,Z 163.163,A -85,B 0,C 180,E1 -6548.995,E2 -6548.995} C_VEL
LIN {X 0,Y 489.487,Z 182.861,A -85,B 0,C 180,E1 -6552.235,E2 -6552.235} C_VEL
LIN {X 0,Y 489.229,Z 192.203,A -85,B 0,C 180,E1 -6553.748,E2 -6553.748} C_VEL
LIN {X 0,Y 491.588,Z 208.988,A -85,B 0,C 180,E1 -6554.077,E2 -6554.077} C_VEL
LIN {X 0,Y 491.061,Z 300.288,A -85,B 0,C 180,E1 -6555.442,E2 -6555.442} C_VEL
LIN {X 0,Y 490.746,Z 313.619,A -85,B 0,C 180,E1 -6555.803,E2 -6555.803} C_VEL
LIN {X 0,Y 490.353,Z 326.388,A -85,B 0,C 180,E1 -6556.32,E2 -6556.32} C_VEL
LIN {X 0,Y 489.953,Z 337.741,A -85,B 0,C 180,E1 -6556.943,E2 -6556.943} C_VEL
LIN {X 0,Y 489.527,Z 349.445,A -85,B 0,C 180,E1 -6557.774,E2 -6557.774} C_VEL
LIN {X 0,Y 489.132,Z 359.972,A -85,B 0,C 180,E1 -6558.71,E2 -6558.71} C_VEL
LIN {X 0,Y 488.785,Z 368.577,A -85,B 0,C 180,E1 -6559.646,E2 -6559.646} C_VEL
LIN {X 0,Y 488.482,Z 376.514,A -85,B 0,C 180,E1 -6560.685,E2 -6560.685} C_VEL
LIN {X 0,Y 488.244,Z 384.269,A -85,B 0,C 180,E1 -6561.932,E2 -6561.932} C_VEL
LIN {X 0,Y 488.09,Z 389.573,A -85,B 0,C 180,E1 -6562.97,E2 -6562.97} C_VEL
LIN {X 0,Y 488.007,Z 394.717,A -85,B 0,C 180,E1 -6564.214,E2 -6564.214} C_VEL
LIN {X 0,Y 487.918,Z 398.707,A -85,B 0,C 180,E1 -6565.456,E2 -6565.456} C_VEL
LIN {X 0,Y 487.965,Z 401.655,A -85,B 0,C 180,E1 -6566.697,E2 -6566.697} C_VEL
LIN {X 0,Y 487.909,Z 403.057,A -85,B 0,C 180,E1 -6567.523,E2 -6567.523} C_VEL
LIN {X 0,Y 487.891,Z 404.056,A -85,B 0,C 180,E1 -6568.349,E2 -6568.349} C_VEL
LIN {X 0,Y 487.827,Z 404.88,A -85,B 0,C 180,E1 -6570,E2 -6570} C_VEL
LIN {X 0,Y 487.891,Z 404.054,A -85,B 0,C 180,E1 -6571.651,E2 -6571.651} C_VEL
LIN {X 0,Y 487.964,Z 401.654,A -85,B 0,C 180,E1 -6573.303,E2 -6573.303} C_VEL
LIN {X 0,Y 487.918,Z 398.704,A -85,B 0,C 180,E1 -6574.544,E2 -6574.544} C_VEL
LIN {X 0,Y 488.006,Z 394.717,A -85,B 0,C 180,E1 -6575.786,E2 -6575.786} C_VEL
LIN {X 0,Y 488.174,Z 388.59,A -85,B 0,C 180,E1 -6577.237,E2 -6577.237} C_VEL
LIN {X 0,Y 488.342,Z 381.893,A -85,B 0,C 180,E1 -6578.483,E2 -6578.483} C_VEL
LIN {X 0,Y 488.617,Z 373.588,A -85,B 0,C 180,E1 -6579.73,E2 -6579.73} C_VEL
LIN {X 0,Y 488.972,Z 365.084,A -85,B 0,C 180,E1 -6580.769,E2 -6580.769} C_VEL
LIN {X 0,Y 489.364,Z 354.579,A -85,B 0,C 180,E1 -6581.809,E2 -6581.809} C_VEL
LIN {X 0,Y 489.761,Z 343.053,A -85,B 0,C 180,E1 -6582.724,E2 -6582.724} C_VEL
LIN {X 0,Y 490.224,Z 330.894,A -85,B 0,C 180,E1 -6583.472,E2 -6583.472} C_VEL
LIN {X 0,Y 490.668,Z 318.562,A -85,B 0,C 180,E1 -6584.04,E2 -6584.04} C_VEL
LIN {X 0,Y 490.984,Z 305.936,A -85,B 0,C 180,E1 -6584.454,E2 -6584.454} C_VEL
LIN {X 0,Y 491.26,Z 292.867,A -85,B 0,C 180,E1 -6584.71,E2 -6584.71} C_VEL
LIN {X 0,Y 491.514,Z 206.829,A -85,B 0,C 180,E1 -6585.991,E2 -6585.991} C_VEL
LIN {X 0,Y 489.231,Z 191.759,A -85,B 0,C 180,E1 -6586.311,E2 -6586.311} C_VEL
LIN {X 0,Y 489.839,Z 172.425,A -85,B 0,C 180,E1 -6589.486,E2 -6589.486} C_VEL
LIN {X 0,Y 490.545,Z 152.794,A -85,B 0,C 180,E1 -6592.757,E2 -6592.757} C_VEL
LIN {X 0,Y 490.583,Z 147.549,A -85,B 0,C 180,E1 -6593.648,E2 -6593.648} C_VEL
LIN {X 0,Y 488.695,Z 137.614,A -85,B 0,C 180,E1 -6595.49,E2 -6595.49} C_VEL
LIN {X 0,Y 488.687,Z 137.613,A -85,B 0,C 180,E1 -6598.685,E2 -6598.685} C_VEL
LIN {X 0,Y 488.692,Z 137.615,A -85,B 0,C 180,E1 -6601.18,E2 -6601.18} C_VEL
LIN {X 0,Y 488.719,Z 137.603,A -85,B 0,C 180,E1 -6604.114,E2 -6604.114} C_VEL
LIN {X 0,Y 488.667,Z 137.614,A -85,B 0,C 180,E1 -6607.16,E2 -6607.16} C_VEL
LIN {X 0,Y 488.696,Z 137.606,A -85,B 0,C 180,E1 -6610.341,E2 -6610.341} C_VEL
LIN {X 0,Y 488.675,Z 137.611,A -85,B 0,C 180,E1 -6613.656,E2 -6613.656} C_VEL
LIN {X 0,Y 488.668,Z 137.611,A -85,B 0,C 180,E1 -6616.343,E2 -6616.343} C_VEL
LIN {X 0,Y 488.669,Z 137.611,A -85,B 0,C 180,E1 -6619.67,E2 -6619.67} C_VEL
LIN {X 0,Y 488.643,Z 137.619,A -85,B 0,C 180,E1 -6622.837,E2 -6622.837} C_VEL
LIN {X 0,Y 488.702,Z 137.604,A -85,B 0,C 180,E1 -6625.884,E2 -6625.884} C_VEL
LIN {X 0,Y 488.66,Z 137.614,A -85,B 0,C 180,E1 -6628.818,E2 -6628.818} C_VEL
LIN {X 0,Y 488.686,Z 137.608,A -85,B 0,C 180,E1 -6631.667,E2 -6631.667} C_VEL
LIN {X 0,Y 488.695,Z 137.609,A -85,B 0,C 180,E1 -6634.961,E2 -6634.961} C_VEL
LIN {X 0,Y 488.684,Z 137.607,A -85,B 0,C 180,E1 -6638.042,E2 -6638.042} C_VEL
LIN {X 0,Y 488.67,Z 137.611,A -85,B 0,C 180,E1 -6640.683,E2 -6640.683} C_VEL
LIN {X 0,Y 488.675,Z 137.608,A -85,B 0,C 180,E1 -6643.283,E2 -6643.283} C_VEL
LIN {X 0,Y 488.72,Z 137.609,A -85,B 0,C 180,E1 -6645.849,E2 -6645.849} C_VEL
LIN {X 0,Y 488.788,Z 137.599,A -85,B 0,C 180,E1 -6648.387,E2 -6648.387} C_VEL
LIN {X 0,Y 488.764,Z 137.6,A -85,B 0,C 180,E1 -6651.732,E2 -6651.732} C_VEL
LIN {X 0,Y 488.818,Z 137.594,A -85,B 0,C 180,E1 -6654.223,E2 -6654.223} C_VEL
LIN {X 0,Y 488.946,Z 137.576,A -85,B 0,C 180,E1 -6657.528,E2 -6657.528} C_VEL
LIN {X 0,Y 488.947,Z 137.576,A -85,B 0,C 180,E1 -6660,E2 -6660} C_VEL
LIN {X 0,Y 488.955,Z 137.573,A -85,B 0,C 180,E1 -6662.471,E2 -6662.471} C_VEL
LIN {X 0,Y 488.832,Z 137.591,A -85,B 0,C 180,E1 -6665.776,E2 -6665.776} C_VEL
LIN {X 0,Y 488.782,Z 137.596,A -85,B 0,C 180,E1 -6668.267,E2 -6668.267} C_VEL
LIN {X 0,Y 488.808,Z 137.597,A -85,B 0,C 180,E1 -6671.612,E2 -6671.612} C_VEL
LIN {X 0,Y 488.761,Z 137.601,A -85,B 0,C 180,E1 -6675,E2 -6675} C_VEL
LIN {X 0,Y 488.747,Z 137.6,A -85,B 0,C 180,E1 -6678.442,E2 -6678.442} C_VEL
LIN {X 0,Y 488.708,Z 137.61,A -85,B 0,C 180,E1 -6681.07,E2 -6681.07} C_VEL
LIN {X 0,Y 488.672,Z 137.611,A -85,B 0,C 180,E1 -6683.746,E2 -6683.746} C_VEL
LIN {X 0,Y 488.749,Z 137.606,A -85,B 0,C 180,E1 -6686.933,E2 -6686.933} C_VEL
LIN {X 0,Y 488.723,Z 137.606,A -85,B 0,C 180,E1 -6689.27,E2 -6689.27} C_VEL
LIN {X 0,Y 488.702,Z 137.61,A -85,B 0,C 180,E1 -6692.147,E2 -6692.147} C_VEL
LIN {X 0,Y 488.714,Z 137.608,A -85,B 0,C 180,E1 -6695.115,E2 -6695.115} C_VEL
LIN {X 0,Y 488.679,Z 137.618,A -85,B 0,C 180,E1 -6698.199,E2 -6698.199} C_VEL
LIN {X 0,Y 488.717,Z 137.615,A -85,B 0,C 180,E1 -6700.344,E2 -6700.344} C_VEL
LIN {X 0,Y 488.686,Z 137.615,A -85,B 0,C 180,E1 -6703.654,E2 -6703.654} C_VEL
LIN {X 0,Y 488.685,Z 137.615,A -85,B 0,C 180,E1 -6706.345,E2 -6706.345} C_VEL
LIN {X 0,Y 488.787,Z 137.625,A -85,B 0,C 180,E1 -6709.523,E2 -6709.523} C_VEL
LIN {X 0,Y 489.74,Z 144.019,A -85,B 0,C 180,E1 -6710.845,E2 -6710.845} C_VEL
LIN {X 0,Y 489.421,Z 158.406,A -85,B 0,C 180,E1 -6713.676,E2 -6713.676} C_VEL
LIN {X 0,Y 489.404,Z 158.836,A -85,B 0,C 180,E1 -6713.761,E2 -6713.761} C_VEL
LIN {X 0,Y 491.918,Z 171.813,A -85,B 0,C 180,E1 -6714.055,E2 -6714.055} C_VEL
LIN {X 0,Y 491.533,Z 219.636,A -85,B 0,C 180,E1 -6714.762,E2 -6714.762} C_VEL
LIN {X 0,Y 490.85,Z 225.478,A -85,B 0,C 180,E1 -6714.826,E2 -6714.826} C_VEL
LIN {X 0,Y 485.251,Z 244.489,A -85,B 0,C 180,E1 -6714.921,E2 -6714.921} C_VEL
LIN {X 0,Y 484.531,Z 250.333,A -85,B 0,C 180,E1 -6714.986,E2 -6714.986} C_VEL
LIN {X 0,Y 484.341,Z 269.159,A -85,B 0,C 180,E1 -6715.314,E2 -6715.314} C_VEL
LIN {X 0,Y 484.11,Z 281.438,A -85,B 0,C 180,E1 -6715.688,E2 -6715.688} C_VEL
LIN {X 0,Y 483.752,Z 293.007,A -85,B 0,C 180,E1 -6716.191,E2 -6716.191} C_VEL
LIN {X 0,Y 483.391,Z 304.146,A -85,B 0,C 180,E1 -6716.837,E2 -6716.837} C_VEL
LIN {X 0,Y 482.964,Z 315.432,A -85,B 0,C 180,E1 -6717.671,E2 -6717.671} C_VEL
LIN {X 0,Y 482.491,Z 325.72,A -85,B 0,C 180,E1 -6718.618,E2 -6718.618} C_VEL
LIN {X 0,Y 482.165,Z 334.143,A -85,B 0,C 180,E1 -6719.568,E2 -6719.568} C_VEL
LIN {X 0,Y 481.768,Z 342.585,A -85,B 0,C 180,E1 -6720.726,E2 -6720.726} C_VEL
LIN {X 0,Y 481.428,Z 349.638,A -85,B 0,C 180,E1 -6721.914,E2 -6721.914} C_VEL
LIN {X 0,Y 481.239,Z 355.279,A -85,B 0,C 180,E1 -6723.081,E2 -6723.081} C_VEL
LIN {X 0,Y 481.055,Z 360.589,A -85,B 0,C 180,E1 -6724.47,E2 -6724.47} C_VEL
LIN {X 0,Y 480.909,Z 364.54,A -85,B 0,C 180,E1 -6725.846,E2 -6725.846} C_VEL
LIN {X 0,Y 480.841,Z 366.992,A -85,B 0,C 180,E1 -6727.044,E2 -6727.044} C_VEL
LIN {X 0,Y 480.756,Z 368.91,A -85,B 0,C 180,E1 -6728.564,E2 -6728.564} C_VEL
LIN {X 0,Y 480.777,Z 369.417,A -85,B 0,C 180,E1 -6729.462,E2 -6729.462} C_VEL
LIN {X 0,Y 480.732,Z 369.46,A -85,B 0,C 180,E1 -6730.352,E2 -6730.352} C_VEL
LIN {X 0,Y 480.769,Z 368.566,A -85,B 0,C 180,E1 -6731.837,E2 -6731.837} C_VEL
LIN {X 0,Y 480.79,Z 366.984,A -85,B 0,C 180,E1 -6733.001,E2 -6733.001} C_VEL
LIN {X 0,Y 480.898,Z 365.27,A -85,B 0,C 180,E1 -6733.879,E2 -6733.879} C_VEL
LIN {X 0,Y 481.04,Z 361.821,A -85,B 0,C 180,E1 -6735.186,E2 -6735.186} C_VEL
LIN {X 0,Y 481.158,Z 357.263,A -85,B 0,C 180,E1 -6736.485,E2 -6736.485} C_VEL
LIN {X 0,Y 481.393,Z 351.417,A -85,B 0,C 180,E1 -6737.785,E2 -6737.785} C_VEL
LIN {X 0,Y 481.671,Z 344.155,A -85,B 0,C 180,E1 -6739.066,E2 -6739.066} C_VEL
LIN {X 0,Y 481.993,Z 335.12,A -85,B 0,C 180,E1 -6740.347,E2 -6740.347} C_VEL
LIN {X 0,Y 482.42,Z 325.791,A -85,B 0,C 180,E1 -6741.412,E2 -6741.412} C_VEL
LIN {X 0,Y 482.899,Z 315.154,A -85,B 0,C 180,E1 -6742.387,E2 -6742.387} C_VEL
LIN {X 0,Y 483.346,Z 303.858,A -85,B 0,C 180,E1 -6743.215,E2 -6743.215} C_VEL
LIN {X 0,Y 483.733,Z 291.778,A -85,B 0,C 180,E1 -6743.901,E2 -6743.901} C_VEL
LIN {X 0,Y 483.983,Z 279.169,A -85,B 0,C 180,E1 -6744.427,E2 -6744.427} C_VEL
LIN {X 0,Y 484.231,Z 265.978,A -85,B 0,C 180,E1 -6744.796,E2 -6744.796} C_VEL
LIN {X 0,Y 484.795,Z 171.255,A -85,B 0,C 180,E1 -6746.234,E2 -6746.234} C_VEL
LIN {X 0,Y 482.324,Z 158.857,A -85,B 0,C 180,E1 -6746.528,E2 -6746.528} C_VEL
LIN {X 0,Y 482.661,Z 145.716,A -85,B 0,C 180,E1 -6749.166,E2 -6749.166} C_VEL
LIN {X 0,Y 482.392,Z 141.67,A -85,B 0,C 180,E1 -6750,E2 -6750} C_VEL
LIN {X 0,Y 481.7,Z 138.484,A -85,B 0,C 180,E1 -6750.706,E2 -6750.706} C_VEL
LIN {X 0,Y 481.901,Z 138.46,A -85,B 0,C 180,E1 -6752.508,E2 -6752.508} C_VEL
LIN {X 0,Y 481.766,Z 138.477,A -85,B 0,C 180,E1 -6755.861,E2 -6755.861} C_VEL
LIN {X 0,Y 481.711,Z 138.478,A -85,B 0,C 180,E1 -6758.389,E2 -6758.389} C_VEL
LIN {X 0,Y 481.731,Z 138.482,A -85,B 0,C 180,E1 -6761.786,E2 -6761.786} C_VEL
LIN {X 0,Y 481.688,Z 138.482,A -85,B 0,C 180,E1 -6765.226,E2 -6765.226} C_VEL
LIN {X 0,Y 481.635,Z 138.486,A -85,B 0,C 180,E1 -6768.725,E2 -6768.725} C_VEL
LIN {X 0,Y 481.617,Z 138.494,A -85,B 0,C 180,E1 -6771.396,E2 -6771.396} C_VEL
LIN {X 0,Y 481.61,Z 138.49,A -85,B 0,C 180,E1 -6774.117,E2 -6774.117} C_VEL
LIN {X 0,Y 481.638,Z 138.49,A -85,B 0,C 180,E1 -6777.115,E2 -6777.115} C_VEL
LIN {X 0,Y 481.596,Z 138.494,A -85,B 0,C 180,E1 -6779.747,E2 -6779.747} C_VEL
LIN {X 0,Y 481.63,Z 138.488,A -85,B 0,C 180,E1 -6782.678,E2 -6782.678} C_VEL
LIN {X 0,Y 481.643,Z 138.493,A -85,B 0,C 180,E1 -6785.202,E2 -6785.202} C_VEL
LIN {X 0,Y 481.623,Z 138.487,A -85,B 0,C 180,E1 -6788.003,E2 -6788.003} C_VEL
LIN {X 0,Y 481.61,Z 138.497,A -85,B 0,C 180,E1 -6791.047,E2 -6791.047} C_VEL
LIN {X 0,Y 481.648,Z 138.486,A -85,B 0,C 180,E1 -6794.459,E2 -6794.459} C_VEL
LIN {X 0,Y 481.611,Z 138.497,A -85,B 0,C 180,E1 -6796.856,E2 -6796.856} C_VEL
LIN {X 0,Y 481.654,Z 138.484,A -85,B 0,C 180,E1 -6800.058,E2 -6800.058} C_VEL
LIN {X 0,Y 481.608,Z 138.49,A -85,B 0,C 180,E1 -6803.38,E2 -6803.38} C_VEL
LIN {X 0,Y 481.671,Z 138.485,A -85,B 0,C 180,E1 -6806.328,E2 -6806.328} C_VEL
LIN {X 0,Y 481.611,Z 138.489,A -85,B 0,C 180,E1 -6809.427,E2 -6809.427} C_VEL
LIN {X 0,Y 481.643,Z 138.488,A -85,B 0,C 180,E1 -6812.165,E2 -6812.165} C_VEL
LIN {X 0,Y 481.668,Z 138.484,A -85,B 0,C 180,E1 -6814.968,E2 -6814.968} C_VEL
LIN {X 0,Y 481.634,Z 138.487,A -85,B 0,C 180,E1 -6817.705,E2 -6817.705} C_VEL
LIN {X 0,Y 481.635,Z 138.493,A -85,B 0,C 180,E1 -6820.391,E2 -6820.391} C_VEL
LIN {X 0,Y 481.613,Z 138.489,A -85,B 0,C 180,E1 -6823.032,E2 -6823.032} C_VEL
LIN {X 0,Y 481.653,Z 138.485,A -85,B 0,C 180,E1 -6825.638,E2 -6825.638} C_VEL
LIN {X 0,Y 481.739,Z 138.48,A -85,B 0,C 180,E1 -6828.215,E2 -6828.215} C_VEL
LIN {X 0,Y 481.716,Z 138.478,A -85,B 0,C 180,E1 -6831.611,E2 -6831.611} C_VEL
LIN {X 0,Y 481.775,Z 138.474,A -85,B 0,C 180,E1 -6834.14,E2 -6834.14} C_VEL
LIN {X 0,Y 481.91,Z 138.455,A -85,B 0,C 180,E1 -6837.493,E2 -6837.493} C_VEL
LIN {X 0,Y 481.914,Z 138.457,A -85,B 0,C 180,E1 -6840,E2 -6840} C_VEL
LIN {X 0,Y 481.91,Z 138.452,A -85,B 0,C 180,E1 -6842.508,E2 -6842.508} C_VEL
LIN {X 0,Y 481.77,Z 138.475,A -85,B 0,C 180,E1 -6845.861,E2 -6845.861} C_VEL
LIN {X 0,Y 481.722,Z 138.475,A -85,B 0,C 180,E1 -6848.389,E2 -6848.389} C_VEL
LIN {X 0,Y 481.757,Z 138.476,A -85,B 0,C 180,E1 -6851.785,E2 -6851.785} C_VEL
LIN {X 0,Y 481.733,Z 138.479,A -85,B 0,C 180,E1 -6855.225,E2 -6855.225} C_VEL
LIN {X 0,Y 481.709,Z 138.478,A -85,B 0,C 180,E1 -6858.722,E2 -6858.722} C_VEL
LIN {X 0,Y 481.642,Z 138.492,A -85,B 0,C 180,E1 -6861.395,E2 -6861.395} C_VEL
LIN {X 0,Y 481.65,Z 138.484,A -85,B 0,C 180,E1 -6864.115,E2 -6864.115} C_VEL
LIN {X 0,Y 481.656,Z 138.491,A -85,B 0,C 180,E1 -6867.117,E2 -6867.117} C_VEL
LIN {X 0,Y 481.656,Z 138.484,A -85,B 0,C 180,E1 -6869.743,E2 -6869.743} C_VEL
LIN {X 0,Y 481.654,Z 138.487,A -85,B 0,C 180,E1 -6872.676,E2 -6872.676} C_VEL
LIN {X 0,Y 481.635,Z 138.486,A -85,B 0,C 180,E1 -6875.71,E2 -6875.71} C_VEL
LIN {X 0,Y 481.67,Z 138.49,A -85,B 0,C 180,E1 -6878.86,E2 -6878.86} C_VEL
LIN {X 0,Y 481.62,Z 138.489,A -85,B 0,C 180,E1 -6882.164,E2 -6882.164} C_VEL
LIN {X 0,Y 481.658,Z 138.488,A -85,B 0,C 180,E1 -6884.458,E2 -6884.458} C_VEL
LIN {X 0,Y 481.62,Z 138.493,A -85,B 0,C 180,E1 -6886.855,E2 -6886.855} C_VEL
LIN {X 0,Y 481.661,Z 138.484,A -85,B 0,C 180,E1 -6890.057,E2 -6890.057} C_VEL
LIN {X 0,Y 481.624,Z 138.488,A -85,B 0,C 180,E1 -6893.252,E2 -6893.252} C_VEL
LIN {X 0,Y 481.674,Z 138.488,A -85,B 0,C 180,E1 -6896.327,E2 -6896.327} C_VEL
LIN {X 0,Y 481.649,Z 138.486,A -85,B 0,C 180,E1 -6899.418,E2 -6899.418} C_VEL
LIN {X 0,Y 481.654,Z 138.493,A -85,B 0,C 180,E1 -6902.165,E2 -6902.165} C_VEL
LIN {X 0,Y 481.695,Z 138.556,A -85,B 0,C 180,E1 -6904.431,E2 -6904.431} C_VEL
LIN {X 0,Y 483.625,Z 148.702,A -85,B 0,C 180,E1 -6906.279,E2 -6906.279} C_VEL
LIN {X 0,Y 483.307,Z 160.193,A -85,B 0,C 180,E1 -6908.235,E2 -6908.235} C_VEL
LIN {X 0,Y 482.564,Z 181.206,A -85,B 0,C 180,E1 -6911.752,E2 -6911.752} C_VEL
LIN {X 0,Y 482.249,Z 191.793,A -85,B 0,C 180,E1 -6913.506,E2 -6913.506} C_VEL
LIN {X 0,Y 484.742,Z 209.725,A -85,B 0,C 180,E1 -6913.868,E2 -6913.868} C_VEL
LIN {X 0,Y 484.177,Z 300.878,A -85,B 0,C 180,E1 -6915.257,E2 -6915.257} C_VEL
LIN {X 0,Y 483.848,Z 313.923,A -85,B 0,C 180,E1 -6915.623,E2 -6915.623} C_VEL
LIN {X 0,Y 483.465,Z 325.983,A -85,B 0,C 180,E1 -6916.122,E2 -6916.122} C_VEL
LIN {X 0,Y 482.99,Z 337.697,A -85,B 0,C 180,E1 -6916.772,E2 -6916.772} C_VEL
LIN {X 0,Y 482.555,Z 349.206,A -85,B 0,C 180,E1 -6917.603,E2 -6917.603} C_VEL
LIN {X 0,Y 482.144,Z 359.645,A -85,B 0,C 180,E1 -6918.544,E2 -6918.544} C_VEL
LIN {X 0,Y 481.745,Z 368.261,A -85,B 0,C 180,E1 -6919.493,E2 -6919.493} C_VEL
LIN {X 0,Y 481.451,Z 376.209,A -85,B 0,C 180,E1 -6920.548,E2 -6920.548} C_VEL
LIN {X 0,Y 481.173,Z 383.976,A -85,B 0,C 180,E1 -6921.813,E2 -6921.813} C_VEL
LIN {X 0,Y 481.017,Z 389.286,A -85,B 0,C 180,E1 -6922.866,E2 -6922.866} C_VEL
LIN {X 0,Y 480.91,Z 394.437,A -85,B 0,C 180,E1 -6924.128,E2 -6924.128} C_VEL
LIN {X 0,Y 480.837,Z 398.433,A -85,B 0,C 180,E1 -6925.389,E2 -6925.389} C_VEL
LIN {X 0,Y 480.888,Z 401.386,A -85,B 0,C 180,E1 -6926.648,E2 -6926.648} C_VEL
LIN {X 0,Y 480.821,Z 403.793,A -85,B 0,C 180,E1 -6928.325,E2 -6928.325} C_VEL
LIN {X 0,Y 480.75,Z 404.622,A -85,B 0,C 180,E1 -6930,E2 -6930} C_VEL
LIN {X 0,Y 480.821,Z 403.8,A -85,B 0,C 180,E1 -6931.675,E2 -6931.675} C_VEL
LIN {X 0,Y 480.888,Z 401.403,A -85,B 0,C 180,E1 -6933.351,E2 -6933.351} C_VEL
LIN {X 0,Y 480.837,Z 398.454,A -85,B 0,C 180,E1 -6934.611,E2 -6934.611} C_VEL
LIN {X 0,Y 480.907,Z 394.469,A -85,B 0,C 180,E1 -6935.871,E2 -6935.871} C_VEL
LIN {X 0,Y 481.102,Z 388.346,A -85,B 0,C 180,E1 -6937.344,E2 -6937.344} C_VEL
LIN {X 0,Y 481.298,Z 381.653,A -85,B 0,C 180,E1 -6938.608,E2 -6938.608} C_VEL
LIN {X 0,Y 481.559,Z 373.351,A -85,B 0,C 180,E1 -6939.874,E2 -6939.874} C_VEL
LIN {X 0,Y 481.972,Z 364.854,A -85,B 0,C 180,E1 -6940.927,E2 -6940.927} C_VEL
LIN {X 0,Y 482.372,Z 354.436,A -85,B 0,C 180,E1 -6941.975,E2 -6941.975} C_VEL
LIN {X 0,Y 482.823,Z 342.695,A -85,B 0,C 180,E1 -6942.921,E2 -6942.921} C_VEL
LIN {X 0,Y 483.31,Z 330.702,A -85,B 0,C 180,E1 -6943.668,E2 -6943.668} C_VEL
LIN {X 0,Y 483.789,Z 318.418,A -85,B 0,C 180,E1 -6944.244,E2 -6944.244} C_VEL
LIN {X 0,Y 484.134,Z 305.883,A -85,B 0,C 180,E1 -6944.663,E2 -6944.663} C_VEL
LIN {X 0,Y 484.425,Z 293.074,A -85,B 0,C 180,E1 -6944.923,E2 -6944.923} C_VEL
LIN {X 0,Y 484.735,Z 207.716,A -85,B 0,C 180,E1 -6946.216,E2 -6946.216} C_VEL
LIN {X 0,Y 482.23,Z 191.518,A -85,B 0,C 180,E1 -6946.565,E2 -6946.565} C_VEL
LIN {X 0,Y 482.907,Z 172.251,A -85,B 0,C 180,E1 -6949.778,E2 -6949.778} C_VEL
LIN {X 0,Y 483.701,Z 152.621,A -85,B 0,C 180,E1 -6953.098,E2 -6953.098} C_VEL
LIN {X 0,Y 483.438,Z 147.38,A -85,B 0,C 180,E1 -6954.02,E2 -6954.02} C_VEL
LIN {X 0,Y 481.67,Z 138.488,A -85,B 0,C 180,E1 -6955.721,E2 -6955.721} C_VEL
LIN {X 0,Y 481.642,Z 138.492,A -85,B 0,C 180,E1 -6958.894,E2 -6958.894} C_VEL
LIN {X 0,Y 481.652,Z 138.487,A -85,B 0,C 180,E1 -6962.187,E2 -6962.187} C_VEL
LIN {X 0,Y 481.658,Z 138.487,A -85,B 0,C 180,E1 -6965.203,E2 -6965.203} C_VEL
LIN {X 0,Y 481.64,Z 138.488,A -85,B 0,C 180,E1 -6968.004,E2 -6968.004} C_VEL
LIN {X 0,Y 481.625,Z 138.489,A -85,B 0,C 180,E1 -6971.045,E2 -6971.045} C_VEL
LIN {X 0,Y 481.655,Z 138.484,A -85,B 0,C 180,E1 -6974.458,E2 -6974.458} C_VEL
LIN {X 0,Y 481.616,Z 138.49,A -85,B 0,C 180,E1 -6977.835,E2 -6977.835} C_VEL
LIN {X 0,Y 481.623,Z 138.492,A -85,B 0,C 180,E1 -6981.136,E2 -6981.136} C_VEL
LIN {X 0,Y 481.609,Z 138.492,A -85,B 0,C 180,E1 -6984.288,E2 -6984.288} C_VEL
LIN {X 0,Y 481.656,Z 138.484,A -85,B 0,C 180,E1 -6986.325,E2 -6986.325} C_VEL
LIN {X 0,Y 481.612,Z 138.487,A -85,B 0,C 180,E1 -6989.426,E2 -6989.426} C_VEL
LIN {X 0,Y 481.644,Z 138.488,A -85,B 0,C 180,E1 -6992.164,E2 -6992.164} C_VEL
LIN {X 0,Y 481.669,Z 138.484,A -85,B 0,C 180,E1 -6994.967,E2 -6994.967} C_VEL
LIN {X 0,Y 481.635,Z 138.482,A -85,B 0,C 180,E1 -6997.704,E2 -6997.704} C_VEL
LIN {X 0,Y 481.624,Z 138.492,A -85,B 0,C 180,E1 -7000.389,E2 -7000.389} C_VEL
LIN {X 0,Y 481.616,Z 138.488,A -85,B 0,C 180,E1 -7003.031,E2 -7003.031} C_VEL
LIN {X 0,Y 481.672,Z 138.484,A -85,B 0,C 180,E1 -7005.638,E2 -7005.638} C_VEL
LIN {X 0,Y 481.739,Z 138.479,A -85,B 0,C 180,E1 -7008.214,E2 -7008.214} C_VEL
LIN {X 0,Y 481.723,Z 138.477,A -85,B 0,C 180,E1 -7011.611,E2 -7011.611} C_VEL
LIN {X 0,Y 481.779,Z 138.472,A -85,B 0,C 180,E1 -7014.139,E2 -7014.139} C_VEL
LIN {X 0,Y 481.911,Z 138.451,A -85,B 0,C 180,E1 -7017.492,E2 -7017.492} C_VEL
LIN {X 0,Y 481.917,Z 138.452,A -85,B 0,C 180,E1 -7020,E2 -7020} C_VEL
LIN {X 0,Y 481.921,Z 138.449,A -85,B 0,C 180,E1 -7022.507,E2 -7022.507} C_VEL
LIN {X 0,Y 481.791,Z 138.467,A -85,B 0,C 180,E1 -7025.86,E2 -7025.86} C_VEL
LIN {X 0,Y 481.738,Z 138.474,A -85,B 0,C 180,E1 -7028.388,E2 -7028.388} C_VEL
LIN {X 0,Y 481.753,Z 138.474,A -85,B 0,C 180,E1 -7031.784,E2 -7031.784} C_VEL
LIN {X 0,Y 481.743,Z 138.478,A -85,B 0,C 180,E1 -7035.224,E2 -7035.224} C_VEL
LIN {X 0,Y 481.709,Z 138.479,A -85,B 0,C 180,E1 -7038.721,E2 -7038.721} C_VEL
LIN {X 0,Y 481.646,Z 138.485,A -85,B 0,C 180,E1 -7041.394,E2 -7041.394} C_VEL
LIN {X 0,Y 481.651,Z 138.486,A -85,B 0,C 180,E1 -7044.114,E2 -7044.114} C_VEL
LIN {X 0,Y 481.716,Z 138.48,A -85,B 0,C 180,E1 -7047.131,E2 -7047.131} C_VEL
LIN {X 0,Y 481.678,Z 138.482,A -85,B 0,C 180,E1 -7049.741,E2 -7049.741} C_VEL
LIN {X 0,Y 481.67,Z 138.488,A -85,B 0,C 180,E1 -7052.674,E2 -7052.674} C_VEL
LIN {X 0,Y 481.635,Z 138.489,A -85,B 0,C 180,E1 -7055.709,E2 -7055.709} C_VEL
LIN {X 0,Y 481.67,Z 138.485,A -85,B 0,C 180,E1 -7058.859,E2 -7058.859} C_VEL
LIN {X 0,Y 481.652,Z 138.491,A -85,B 0,C 180,E1 -7061.912,E2 -7061.912} C_VEL
LIN {X 0,Y 481.658,Z 138.49,A -85,B 0,C 180,E1 -7064.457,E2 -7064.457} C_VEL
LIN {X 0,Y 481.647,Z 138.492,A -85,B 0,C 180,E1 -7067.839,E2 -7067.839} C_VEL
LIN {X 0,Y 481.735,Z 138.528,A -85,B 0,C 180,E1 -7069.342,E2 -7069.342} C_VEL
LIN {X 0,Y 482.794,Z 145.921,A -85,B 0,C 180,E1 -7070.883,E2 -7070.883} C_VEL
LIN {X 0,Y 482.464,Z 159.008,A -85,B 0,C 180,E1 -7073.491,E2 -7073.491} C_VEL
LIN {X 0,Y 485.169,Z 173.118,A -85,B 0,C 180,E1 -7073.826,E2 -7073.826} C_VEL
LIN {X 0,Y 484.531,Z 250.333,A -85,B 0,C 180,E1 -7074.986,E2 -7074.986} C_VEL
LIN {X 0,Y 483.743,Z 256.186,A -85,B 0,C 180,E1 -7075.046,E2 -7075.046} C_VEL
LIN {X 0,Y 480.713,Z 265.665,A -85,B 0,C 180,E1 -7075.105,E2 -7075.105} C_VEL
LIN {X 0,Y 477.879,Z 275.108,A -85,B 0,C 180,E1 -7075.255,E2 -7075.255} C_VEL
LIN {X 0,Y 477.288,Z 280.718,A -85,B 0,C 180,E1 -7075.427,E2 -7075.427} C_VEL
LIN {X 0,Y 476.925,Z 292.746,A -85,B 0,C 180,E1 -7075.946,E2 -7075.946} C_VEL
LIN {X 0,Y 476.486,Z 305.077,A -85,B 0,C 180,E1 -7076.672,E2 -7076.672} C_VEL
LIN {X 0,Y 476.047,Z 316.092,A -85,B 0,C 180,E1 -7077.506,E2 -7077.506} C_VEL
LIN {X 0,Y 475.542,Z 326.423,A -85,B 0,C 180,E1 -7078.479,E2 -7078.479} C_VEL
LIN {X 0,Y 475.12,Z 335.754,A -85,B 0,C 180,E1 -7079.574,E2 -7079.574} C_VEL
LIN {X 0,Y 474.7,Z 344.672,A -85,B 0,C 180,E1 -7080.867,E2 -7080.867} C_VEL
LIN {X 0,Y 474.331,Z 351.931,A -85,B 0,C 180,E1 -7082.178,E2 -7082.178} C_VEL
LIN {X 0,Y 474.102,Z 358.068,A -85,B 0,C 180,E1 -7083.595,E2 -7083.595} C_VEL
LIN {X 0,Y 473.934,Z 362.071,A -85,B 0,C 180,E1 -7084.764,E2 -7084.764} C_VEL
LIN {X 0,Y 473.793,Z 366.145,A -85,B 0,C 180,E1 -7086.39,E2 -7086.39} C_VEL
LIN {X 0,Y 473.717,Z 367.78,A -85,B 0,C 180,E1 -7087.311,E2 -7087.311} C_VEL
LIN {X 0,Y 473.663,Z 368.883,A -85,B 0,C 180,E1 -7088.226,E2 -7088.226} C_VEL
LIN {X 0,Y 473.677,Z 369.572,A -85,B 0,C 180,E1 -7089.184,E2 -7089.184} C_VEL
LIN {X 0,Y 473.664,Z 369.775,A -85,B 0,C 180,E1 -7090.046,E2 -7090.046} C_VEL
LIN {X 0,Y 473.682,Z 368.951,A -85,B 0,C 180,E1 -7091.724,E2 -7091.724} C_VEL
LIN {X 0,Y 473.704,Z 367.741,A -85,B 0,C 180,E1 -7092.739,E2 -7092.739} C_VEL
LIN {X 0,Y 473.843,Z 365.221,A -85,B 0,C 180,E1 -7094.074,E2 -7094.074} C_VEL
LIN {X 0,Y 473.985,Z 361.654,A -85,B 0,C 180,E1 -7095.4,E2 -7095.4} C_VEL
LIN {X 0,Y 474.103,Z 356.96,A -85,B 0,C 180,E1 -7096.717,E2 -7096.717} C_VEL
LIN {X 0,Y 474.337,Z 350.979,A -85,B 0,C 180,E1 -7098.028,E2 -7098.028} C_VEL
LIN {X 0,Y 474.674,Z 343.512,A -85,B 0,C 180,E1 -7099.335,E2 -7099.335} C_VEL
LIN {X 0,Y 474.972,Z 335.925,A -85,B 0,C 180,E1 -7100.418,E2 -7100.418} C_VEL
LIN {X 0,Y 475.42,Z 326.714,A -85,B 0,C 180,E1 -7101.499,E2 -7101.499} C_VEL
LIN {X 0,Y 475.908,Z 316.47,A -85,B 0,C 180,E1 -7102.469,E2 -7102.469} C_VEL
LIN {X 0,Y 476.38,Z 305.105,A -85,B 0,C 180,E1 -7103.328,E2 -7103.328} C_VEL
LIN {X 0,Y 476.741,Z 293.374,A -85,B 0,C 180,E1 -7104.024,E2 -7104.024} C_VEL
LIN {X 0,Y 477.067,Z 280.505,A -85,B 0,C 180,E1 -7104.585,E2 -7104.585} C_VEL
LIN {X 0,Y 477.335,Z 267.81,A -85,B 0,C 180,E1 -7104.958,E2 -7104.958} C_VEL
LIN {X 0,Y 477.564,Z 238.422,A -85,B 0,C 180,E1 -7105.437,E2 -7105.437} C_VEL
LIN {X 0,Y 477.993,Z 172.369,A -85,B 0,C 180,E1 -7106.444,E2 -7106.444} C_VEL
LIN {X 0,Y 475.364,Z 159.17,A -85,B 0,C 180,E1 -7106.742,E2 -7106.742} C_VEL
LIN {X 0,Y 475.682,Z 146.252,A -85,B 0,C 180,E1 -7109.365,E2 -7109.365} C_VEL
LIN {X 0,Y 475.043,Z 141.238,A -85,B 0,C 180,E1 -7110.424,E2 -7110.424} C_VEL
LIN {X 0,Y 474.65,Z 139.362,A -85,B 0,C 180,E1 -7110.849,E2 -7110.849} C_VEL
LIN {X 0,Y 474.866,Z 139.336,A -85,B 0,C 180,E1 -7112.545,E2 -7112.545} C_VEL
LIN {X 0,Y 474.73,Z 139.354,A -85,B 0,C 180,E1 -7115.948,E2 -7115.948} C_VEL
LIN {X 0,Y 474.659,Z 139.356,A -85,B 0,C 180,E1 -7118.515,E2 -7118.515} C_VEL
LIN {X 0,Y 474.688,Z 139.357,A -85,B 0,C 180,E1 -7121.963,E2 -7121.963} C_VEL
LIN {X 0,Y 474.646,Z 139.361,A -85,B 0,C 180,E1 -7125.458,E2 -7125.458} C_VEL
LIN {X 0,Y 474.588,Z 139.365,A -85,B 0,C 180,E1 -7129.014,E2 -7129.014} C_VEL
LIN {X 0,Y 474.565,Z 139.372,A -85,B 0,C 180,E1 -7131.73,E2 -7131.73} C_VEL
LIN {X 0,Y 474.577,Z 139.365,A -85,B 0,C 180,E1 -7134.498,E2 -7134.498} C_VEL
LIN {X 0,Y 474.589,Z 139.371,A -85,B 0,C 180,E1 -7137.327,E2 -7137.327} C_VEL
LIN {X 0,Y 474.545,Z 139.369,A -85,B 0,C 180,E1 -7140.235,E2 -7140.235} C_VEL
LIN {X 0,Y 474.604,Z 139.37,A -85,B 0,C 180,E1 -7143.224,E2 -7143.224} C_VEL
LIN {X 0,Y 474.566,Z 139.367,A -85,B 0,C 180,E1 -7146.326,E2 -7146.326} C_VEL
LIN {X 0,Y 474.599,Z 139.365,A -85,B 0,C 180,E1 -7149.551,E2 -7149.551} C_VEL
LIN {X 0,Y 474.573,Z 139.366,A -85,B 0,C 180,E1 -7152.231,E2 -7152.231} C_VEL
LIN {X 0,Y 474.611,Z 139.364,A -85,B 0,C 180,E1 -7155.299,E2 -7155.299} C_VEL
LIN {X 0,Y 474.59,Z 139.364,A -85,B 0,C 180,E1 -7158.212,E2 -7158.212} C_VEL
LIN {X 0,Y 474.617,Z 139.363,A -85,B 0,C 180,E1 -7160.452,E2 -7160.452} C_VEL
LIN {X 0,Y 474.571,Z 139.366,A -85,B 0,C 180,E1 -7163.676,E2 -7163.676} C_VEL
LIN {X 0,Y 474.608,Z 139.368,A -85,B 0,C 180,E1 -7166.778,E2 -7166.778} C_VEL
LIN {X 0,Y 474.55,Z 139.369,A -85,B 0,C 180,E1 -7169.767,E2 -7169.767} C_VEL
LIN {X 0,Y 474.602,Z 139.368,A -85,B 0,C 180,E1 -7172.685,E2 -7172.685} C_VEL
LIN {X 0,Y 474.587,Z 139.364,A -85,B 0,C 180,E1 -7175.504,E2 -7175.504} C_VEL
LIN {X 0,Y 474.596,Z 139.365,A -85,B 0,C 180,E1 -7178.898,E2 -7178.898} C_VEL
LIN {X 0,Y 474.612,Z 139.364,A -85,B 0,C 180,E1 -7181.883,E2 -7181.883} C_VEL
LIN {X 0,Y 474.653,Z 139.359,A -85,B 0,C 180,E1 -7184.543,E2 -7184.543} C_VEL
LIN {X 0,Y 474.697,Z 139.357,A -85,B 0,C 180,E1 -7188.038,E2 -7188.038} C_VEL
LIN {X 0,Y 474.665,Z 139.356,A -85,B 0,C 180,E1 -7191.486,E2 -7191.486} C_VEL
LIN {X 0,Y 474.739,Z 139.352,A -85,B 0,C 180,E1 -7194.052,E2 -7194.052} C_VEL
LIN {X 0,Y 474.875,Z 139.331,A -85,B 0,C 180,E1 -7197.456,E2 -7197.456} C_VEL
LIN {X 0,Y 474.884,Z 139.333,A -85,B 0,C 180,E1 -7200,E2 -7200} C_VEL
LIN {X 0,Y 474.875,Z 139.328,A -85,B 0,C 180,E1 -7202.545,E2 -7202.545} C_VEL
LIN {X 0,Y 474.733,Z 139.35,A -85,B 0,C 180,E1 -7205.949,E2 -7205.949} C_VEL
LIN {X 0,Y 474.671,Z 139.353,A -85,B 0,C 180,E1 -7208.515,E2 -7208.515} C_VEL
LIN {X 0,Y 474.71,Z 139.351,A -85,B 0,C 180,E1 -7211.963,E2 -7211.963} C_VEL
LIN {X 0,Y 474.657,Z 139.359,A -85,B 0,C 180,E1 -7215.755,E2 -7215.755} C_VEL
LIN {X 0,Y 474.662,Z 139.358,A -85,B 0,C 180,E1 -7219.011,E2 -7219.011} C_VEL
LIN {X 0,Y 474.585,Z 139.367,A -85,B 0,C 180,E1 -7221.73,E2 -7221.73} C_VEL
LIN {X 0,Y 474.629,Z 139.359,A -85,B 0,C 180,E1 -7224.495,E2 -7224.495} C_VEL
LIN {X 0,Y 474.603,Z 139.368,A -85,B 0,C 180,E1 -7227.326,E2 -7227.326} C_VEL
LIN {X 0,Y 474.585,Z 139.364,A -85,B 0,C 180,E1 -7230.232,E2 -7230.232} C_VEL
LIN {X 0,Y 474.618,Z 139.365,A -85,B 0,C 180,E1 -7233.222,E2 -7233.222} C_VEL
LIN {X 0,Y 474.588,Z 139.365,A -85,B 0,C 180,E1 -7236.324,E2 -7236.324} C_VEL
LIN {X 0,Y 474.626,Z 139.36,A -85,B 0,C 180,E1 -7239.548,E2 -7239.548} C_VEL
LIN {X 0,Y 474.58,Z 139.366,A -85,B 0,C 180,E1 -7242.23,E2 -7242.23} C_VEL
LIN {X 0,Y 474.62,Z 139.361,A -85,B 0,C 180,E1 -7245.298,E2 -7245.298} C_VEL
LIN {X 0,Y 474.596,Z 139.365,A -85,B 0,C 180,E1 -7248.211,E2 -7248.211} C_VEL
LIN {X 0,Y 474.612,Z 139.361,A -85,B 0,C 180,E1 -7251.542,E2 -7251.542} C_VEL
LIN {X 0,Y 474.623,Z 139.364,A -85,B 0,C 180,E1 -7254.725,E2 -7254.725} C_VEL
LIN {X 0,Y 474.631,Z 139.36,A -85,B 0,C 180,E1 -7257.787,E2 -7257.787} C_VEL
LIN {X 0,Y 474.602,Z 139.366,A -85,B 0,C 180,E1 -7260.89,E2 -7260.89} C_VEL
LIN {X 0,Y 474.665,Z 139.492,A -85,B 0,C 180,E1 -7264.263,E2 -7264.263} C_VEL
LIN {X 0,Y 476.683,Z 150.212,A -85,B 0,C 180,E1 -7266.239,E2 -7266.239} C_VEL
LIN {X 0,Y 476.239,Z 165.156,A -85,B 0,C 180,E1 -7268.811,E2 -7268.811} C_VEL
LIN {X 0,Y 475.442,Z 184.797,A -85,B 0,C 180,E1 -7272.138,E2 -7272.138} C_VEL
LIN {X 0,Y 475.241,Z 191.589,A -85,B 0,C 180,E1 -7273.28,E2 -7273.28} C_VEL
LIN {X 0,Y 477.91,Z 210.971,A -85,B 0,C 180,E1 -7273.669,E2 -7273.669} C_VEL
LIN {X 0,Y 477.29,Z 300.096,A -85,B 0,C 180,E1 -7275.04,E2 -7275.04} C_VEL
LIN {X 0,Y 476.948,Z 313.334,A -85,B 0,C 180,E1 -7275.411,E2 -7275.411} C_VEL
LIN {X 0,Y 476.551,Z 325.499,A -85,B 0,C 180,E1 -7275.916,E2 -7275.916} C_VEL
LIN {X 0,Y 476.064,Z 336.966,A -85,B 0,C 180,E1 -7276.555,E2 -7276.555} C_VEL
LIN {X 0,Y 475.606,Z 348.518,A -85,B 0,C 180,E1 -7277.391,E2 -7277.391} C_VEL
LIN {X 0,Y 475.162,Z 359.318,A -85,B 0,C 180,E1 -7278.374,E2 -7278.374} C_VEL
LIN {X 0,Y 474.733,Z 367.945,A -85,B 0,C 180,E1 -7279.336,E2 -7279.336} C_VEL
LIN {X 0,Y 474.433,Z 375.904,A -85,B 0,C 180,E1 -7280.407,E2 -7280.407} C_VEL
LIN {X 0,Y 474.129,Z 383.683,A -85,B 0,C 180,E1 -7281.69,E2 -7281.69} C_VEL
LIN {X 0,Y 473.897,Z 390.832,A -85,B 0,C 180,E1 -7283.186,E2 -7283.186} C_VEL
LIN {X 0,Y 473.836,Z 395.596,A -85,B 0,C 180,E1 -7284.467,E2 -7284.467} C_VEL
LIN {X 0,Y 473.734,Z 399.233,A -85,B 0,C 180,E1 -7285.746,E2 -7285.746} C_VEL
LIN {X 0,Y 473.795,Z 401.116,A -85,B 0,C 180,E1 -7286.598,E2 -7286.598} C_VEL
LIN {X 0,Y 473.742,Z 402.525,A -85,B 0,C 180,E1 -7287.449,E2 -7287.449} C_VEL
LIN {X 0,Y 473.725,Z 403.528,A -85,B 0,C 180,E1 -7288.3,E2 -7288.3} C_VEL
LIN {X 0,Y 473.677,Z 404.363,A -85,B 0,C 180,E1 -7290,E2 -7290} C_VEL
LIN {X 0,Y 473.693,Z 404.152,A -85,B 0,C 180,E1 -7290.85,E2 -7290.85} C_VEL
LIN {X 0,Y 473.725,Z 403.545,A -85,B 0,C 180,E1 -7291.7,E2 -7291.7} C_VEL
LIN {X 0,Y 473.795,Z 401.15,A -85,B 0,C 180,E1 -7293.401,E2 -7293.401} C_VEL
LIN {X 0,Y 473.76,Z 398.204,A -85,B 0,C 180,E1 -7294.68,E2 -7294.68} C_VEL
LIN {X 0,Y 473.811,Z 394.22,A -85,B 0,C 180,E1 -7295.96,E2 -7295.96} C_VEL
LIN {X 0,Y 474.011,Z 388.102,A -85,B 0,C 180,E1 -7297.454,E2 -7297.454} C_VEL
LIN {X 0,Y 474.246,Z 381.412,A -85,B 0,C 180,E1 -7298.737,E2 -7298.737} C_VEL
LIN {X 0,Y 474.523,Z 373.126,A -85,B 0,C 180,E1 -7300.022,E2 -7300.022} C_VEL
LIN {X 0,Y 474.969,Z 364.657,A -85,B 0,C 180,E1 -7301.09,E2 -7301.09} C_VEL
LIN {X 0,Y 475.388,Z 354.493,A -85,B 0,C 180,E1 -7302.135,E2 -7302.135} C_VEL
LIN {X 0,Y 475.892,Z 342.599,A -85,B 0,C 180,E1 -7303.113,E2 -7303.113} C_VEL
LIN {X 0,Y 476.414,Z 330.708,A -85,B 0,C 180,E1 -7303.87,E2 -7303.87} C_VEL
LIN {X 0,Y 476.916,Z 318.52,A -85,B 0,C 180,E1 -7304.454,E2 -7304.454} C_VEL
LIN {X 0,Y 477.285,Z 306.135,A -85,B 0,C 180,E1 -7304.878,E2 -7304.878} C_VEL
LIN {X 0,Y 477.597,Z 293.813,A -85,B 0,C 180,E1 -7305.141,E2 -7305.141} C_VEL
LIN {X 0,Y 477.974,Z 208.815,A -85,B 0,C 180,E1 -7306.447,E2 -7306.447} C_VEL
LIN {X 0,Y 475.266,Z 191.183,A -85,B 0,C 180,E1 -7306.843,E2 -7306.843} C_VEL
LIN {X 0,Y 475.949,Z 173.387,A -85,B 0,C 180,E1 -7309.854,E2 -7309.854} C_VEL
LIN {X 0,Y 476.778,Z 153.799,A -85,B 0,C 180,E1 -7313.223,E2 -7313.223} C_VEL
LIN {X 0,Y 476.56,Z 148.97,A -85,B 0,C 180,E1 -7314.088,E2 -7314.088} C_VEL
LIN {X 0,Y 474.635,Z 139.365,A -85,B 0,C 180,E1 -7315.93,E2 -7315.93} C_VEL
LIN {X 0,Y 474.603,Z 139.371,A -85,B 0,C 180,E1 -7319.253,E2 -7319.253} C_VEL
LIN {X 0,Y 474.604,Z 139.364,A -85,B 0,C 180,E1 -7322.428,E2 -7322.428} C_VEL
LIN {X 0,Y 474.61,Z 139.368,A -85,B 0,C 180,E1 -7325.468,E2 -7325.468} C_VEL
LIN {X 0,Y 474.594,Z 139.365,A -85,B 0,C 180,E1 -7328.459,E2 -7328.459} C_VEL
LIN {X 0,Y 474.601,Z 139.363,A -85,B 0,C 180,E1 -7330.955,E2 -7330.955} C_VEL
LIN {X 0,Y 474.603,Z 139.362,A -85,B 0,C 180,E1 -7334.106,E2 -7334.106} C_VEL
LIN {X 0,Y 474.568,Z 139.373,A -85,B 0,C 180,E1 -7337.06,E2 -7337.06} C_VEL
LIN {X 0,Y 474.573,Z 139.37,A -85,B 0,C 180,E1 -7339.337,E2 -7339.337} C_VEL
LIN {X 0,Y 474.586,Z 139.364,A -85,B 0,C 180,E1 -7341.708,E2 -7341.708} C_VEL
LIN {X 0,Y 474.602,Z 139.368,A -85,B 0,C 180,E1 -7344.723,E2 -7344.723} C_VEL
LIN {X 0,Y 474.611,Z 139.361,A -85,B 0,C 180,E1 -7347.785,E2 -7347.785} C_VEL
LIN {X 0,Y 474.577,Z 139.369,A -85,B 0,C 180,E1 -7350.895,E2 -7350.895} C_VEL
LIN {X 0,Y 474.574,Z 139.362,A -85,B 0,C 180,E1 -7353.623,E2 -7353.623} C_VEL
LIN {X 0,Y 474.6,Z 139.362,A -85,B 0,C 180,E1 -7356.652,E2 -7356.652} C_VEL
LIN {X 0,Y 474.618,Z 139.36,A -85,B 0,C 180,E1 -7359.183,E2 -7359.183} C_VEL
LIN {X 0,Y 474.612,Z 139.362,A -85,B 0,C 180,E1 -7361.882,E2 -7361.882} C_VEL
LIN {X 0,Y 474.691,Z 139.355,A -85,B 0,C 180,E1 -7364.544,E2 -7364.544} C_VEL
LIN {X 0,Y 474.696,Z 139.354,A -85,B 0,C 180,E1 -7368.037,E2 -7368.037} C_VEL
LIN {X 0,Y 474.698,Z 139.351,A -85,B 0,C 180,E1 -7371.486,E2 -7371.486} C_VEL
LIN {X 0,Y 474.742,Z 139.35,A -85,B 0,C 180,E1 -7374.051,E2 -7374.051} C_VEL
LIN {X 0,Y 474.876,Z 139.327,A -85,B 0,C 180,E1 -7377.455,E2 -7377.455} C_VEL
LIN {X 0,Y 474.886,Z 139.328,A -85,B 0,C 180,E1 -7380,E2 -7380} C_VEL
LIN {X 0,Y 474.887,Z 139.325,A -85,B 0,C 180,E1 -7382.544,E2 -7382.544} C_VEL
LIN {X 0,Y 474.752,Z 139.343,A -85,B 0,C 180,E1 -7385.947,E2 -7385.947} C_VEL
LIN {X 0,Y 474.711,Z 139.349,A -85,B 0,C 180,E1 -7388.513,E2 -7388.513} C_VEL
LIN {X 0,Y 474.707,Z 139.351,A -85,B 0,C 180,E1 -7391.962,E2 -7391.962} C_VEL
LIN {X 0,Y 474.701,Z 139.355,A -85,B 0,C 180,E1 -7395.455,E2 -7395.455} C_VEL
LIN {X 0,Y 474.663,Z 139.359,A -85,B 0,C 180,E1 -7399.01,E2 -7399.01} C_VEL
LIN {X 0,Y 474.589,Z 139.362,A -85,B 0,C 180,E1 -7401.728,E2 -7401.728} C_VEL
LIN {X 0,Y 474.63,Z 139.364,A -85,B 0,C 180,E1 -7404.494,E2 -7404.494} C_VEL
LIN {X 0,Y 474.673,Z 139.355,A -85,B 0,C 180,E1 -7407.332,E2 -7407.332} C_VEL
LIN {X 0,Y 474.604,Z 139.366,A -85,B 0,C 180,E1 -7410.23,E2 -7410.23} C_VEL
LIN {X 0,Y 474.624,Z 139.362,A -85,B 0,C 180,E1 -7413.221,E2 -7413.221} C_VEL
LIN {X 0,Y 474.588,Z 139.372,A -85,B 0,C 180,E1 -7416.323,E2 -7416.323} C_VEL
LIN {X 0,Y 474.626,Z 139.362,A -85,B 0,C 180,E1 -7419.647,E2 -7419.647} C_VEL
LIN {X 0,Y 474.614,Z 139.368,A -85,B 0,C 180,E1 -7422.934,E2 -7422.934} C_VEL
